C05484=1146.169,25.527,-49.640,179.957,6.278,149.150
C05485=1146.174,25.277,-49.625,179.955,6.277,149.150
C05486=1146.179,25.027,-49.611,179.952,6.277,149.151
C05487=1146.184,24.778,-49.597,179.949,6.275,149.151
C05488=1146.190,24.528,-49.582,179.947,6.275,149.152
C05489=1146.195,24.278,-49.568,179.945,6.274,149.152
C05490=1146.200,24.029,-49.554,179.941,6.272,149.153
C05491=1146.205,23.780,-49.539,179.939,6.272,149.154
C05492=1146.210,23.530,-49.525,179.937,6.271,149.154
C05493=1146.215,23.280,-49.510,179.934,6.270,149.155
C05494=1146.220,23.031,-49.496,179.932,6.269,149.155
C05495=1146.225,22.782,-49.482,179.929,6.268,149.156
C05496=1146.230,22.532,-49.468,179.927,6.267,149.156
C05497=1146.235,22.282,-49.454,179.924,6.266,149.157
C05498=1146.240,22.033,-49.439,179.921,6.265,149.157
C05499=1146.245,21.783,-49.425,179.919,6.265,149.158
C05500=1146.251,21.534,-49.411,179.916,6.263,149.159
C05501=1146.256,21.284,-49.397,179.914,6.262,149.159
C05502=1146.261,21.034,-49.382,179.911,6.262,149.160
C05503=1146.266,20.785,-49.368,179.908,6.260,149.160
C05504=1146.271,20.536,-49.354,179.906,6.260,149.161
C05505=1146.276,20.286,-49.340,179.904,6.259,149.161
C05506=1146.281,20.036,-49.326,179.901,6.257,149.162
C05507=1146.286,19.787,-49.311,179.898,6.257,149.162
C05508=1146.291,19.538,-49.298,179.896,6.256,149.163
C05509=1146.296,19.288,-49.283,179.893,6.256,149.164
C05510=1146.301,19.038,-49.269,179.891,6.254,149.164
C05511=1146.306,18.789,-49.255,179.888,6.253,149.164
C05512=1146.312,18.539,-49.241,179.886,6.253,149.165
C05513=1146.316,18.290,-49.227,179.883,6.251,149.166
C05514=1146.321,18.040,-49.214,179.880,6.251,149.166
C05515=1146.326,17.790,-49.199,179.878,6.250,149.167
C05516=1146.332,17.541,-49.185,179.876,6.250,149.167
C05517=1146.337,17.291,-49.171,179.873,6.248,149.168
C05518=1146.342,17.042,-49.157,179.871,6.247,149.168
C05519=1146.347,16.793,-49.143,179.868,6.247,149.169
C05520=1146.352,16.543,-49.129,179.865,6.245,149.169
C05521=1146.358,16.293,-49.115,179.863,6.245,149.170
C05522=1146.362,16.044,-49.102,179.860,6.244,149.171
C05523=1146.367,15.794,-49.087,179.858,6.243,149.171
C05524=1146.372,15.544,-49.073,179.855,6.242,149.172
C05525=1146.377,15.295,-49.059,179.853,6.241,149.172
C05526=1146.383,15.046,-49.045,179.850,6.240,149.173
C05527=1146.388,14.795,-49.031,179.848,6.240,149.173
C05528=1146.393,14.546,-49.017,179.845,6.238,149.174
C05529=1146.398,14.297,-49.004,179.843,6.238,149.174
C05530=1146.403,14.047,-48.990,179.840,6.237,149.175
C05531=1146.409,13.798,-48.976,179.838,6.236,149.176
C05532=1146.414,13.548,-48.962,179.835,6.235,149.176
C05533=1146.419,13.298,-48.948,179.832,6.234,149.177
C05534=1146.423,13.050,-48.935,179.830,6.233,149.177
C05535=1146.429,12.799,-48.921,179.827,6.233,149.178
C05536=1146.434,12.549,-48.907,179.825,6.231,149.178
C05537=1146.439,12.300,-48.893,179.822,6.231,149.179
C05538=1146.444,12.050,-48.879,179.820,6.230,149.180
C05539=1146.449,11.801,-48.866,179.818,6.229,149.180
C05540=1146.454,11.552,-48.852,179.814,6.228,149.181
C05541=1146.459,11.301,-48.838,179.812,6.227,149.181
C05542=1146.465,11.052,-48.824,179.810,6.227,149.182
C05543=1146.469,10.803,-48.810,179.807,6.226,149.182
C05544=1146.474,10.553,-48.797,179.804,6.225,149.183
C05545=1146.480,10.304,-48.783,179.802,6.224,149.183
C05546=1146.485,10.054,-48.770,179.799,6.223,149.184
C05547=1146.490,9.805,-48.756,179.797,6.223,149.185
C05548=1146.495,9.555,-48.742,179.794,6.221,149.185
C05549=1146.501,9.305,-48.729,179.792,6.221,149.186
C05550=1146.505,9.056,-48.715,179.790,6.220,149.186
C05551=1146.510,8.806,-48.701,179.787,6.219,149.187
C05552=1146.516,8.557,-48.687,179.785,6.218,149.187
C05553=1146.520,8.307,-48.675,179.782,6.217,149.188
C05554=1146.526,8.058,-48.661,179.779,6.216,149.188
C05555=1146.531,7.808,-48.646,179.777,6.216,149.189
C05556=1146.536,7.559,-48.634,179.775,6.215,149.190
C05557=1146.541,7.309,-48.619,179.772,6.214,149.190
C05558=1146.547,7.059,-48.606,179.769,6.213,149.191
C05559=1146.551,6.810,-48.593,179.767,6.212,149.191
C05560=1146.557,6.560,-48.579,179.764,6.212,149.192
C05561=1146.561,6.311,-48.566,179.762,6.211,149.192
C05562=1146.567,6.060,-48.552,179.759,6.209,149.193
C05563=1146.572,5.811,-48.538,179.757,6.209,149.194
C05564=1146.577,5.561,-48.525,179.754,6.208,149.194
C05565=1146.582,5.312,-48.512,179.752,6.208,149.195
C05566=1146.587,5.062,-48.498,179.750,6.207,149.195
C05567=1146.593,4.813,-48.485,179.746,6.206,149.196
C05568=1146.597,4.563,-48.471,179.744,6.205,149.196
C05569=1146.603,4.314,-48.458,179.742,6.204,149.197
C05570=1146.608,4.064,-48.444,179.739,6.204,149.197
C05571=1146.613,3.815,-48.431,179.737,6.203,149.198
C05572=1146.618,3.564,-48.418,179.734,6.202,149.199
C05573=1146.623,3.316,-48.405,179.732,6.201,149.199
C05574=1146.629,3.066,-48.391,179.729,6.200,149.200
C05575=1146.634,2.816,-48.378,179.727,6.199,149.200
C05576=1146.639,2.567,-48.364,179.724,6.199,149.201
C05577=1146.644,2.317,-48.351,179.722,6.198,149.201
C05578=1146.649,2.067,-48.338,179.719,6.197,149.202
C05579=1146.655,1.798,-48.323,179.717,6.196,149.202
C05580=1146.660,1.528,-48.309,179.714,6.196,149.203
C05581=1146.666,1.259,-48.295,179.711,6.194,149.204
C05582=1146.671,0.989,-48.281,179.709,6.194,149.204
C05583=1146.676,0.740,-48.267,179.706,6.193,149.205
C05584=1146.681,0.490,-48.254,179.704,6.192,149.205
C05585=1146.686,0.241,-48.241,179.701,6.191,149.206
C05586=1146.691,-0.009,-48.227,179.698,6.190,149.207
C05587=1146.697,-0.258,-48.214,179.696,6.190,149.207
C05588=1146.702,-0.508,-48.201,179.694,6.189,149.208
C05589=1146.707,-0.758,-48.188,179.691,6.188,149.208
C05590=1146.712,-1.007,-48.174,179.689,6.188,149.209
C05591=1146.717,-1.257,-48.161,179.686,6.186,149.209
C05592=1146.723,-1.506,-48.148,179.684,6.186,149.210
C05593=1146.727,-1.756,-48.135,179.681,6.185,149.211
C05594=1146.733,-2.006,-48.123,179.679,6.184,149.211
C05595=1146.738,-2.255,-48.109,179.676,6.184,149.212
C05596=1146.743,-2.505,-48.096,179.674,6.183,149.212
C05597=1146.748,-2.754,-48.082,179.671,6.183,149.213
C05598=1146.753,-3.004,-48.070,179.669,6.181,149.213
C05599=1146.758,-3.254,-48.057,179.666,6.180,149.214
C05600=1146.764,-3.503,-48.044,179.664,6.180,149.214
C05601=1146.769,-3.753,-48.031,179.662,6.179,149.215
C05602=1146.774,-4.002,-48.017,179.659,6.179,149.216
C05603=1146.779,-4.252,-48.004,179.657,6.178,149.216
C05604=1146.784,-4.502,-47.991,179.654,6.177,149.217
C05605=1146.790,-4.751,-47.978,179.651,6.176,149.217
C05606=1146.795,-5.000,-47.965,179.649,6.175,149.218
C05607=1146.799,-5.251,-47.953,179.647,6.174,149.218
C05608=1146.805,-5.500,-47.939,179.644,6.174,149.219
C05609=1146.810,-5.749,-47.927,179.642,6.173,149.220
C05610=1146.815,-5.999,-47.914,179.640,6.172,149.220
C05611=1146.821,-6.249,-47.901,179.637,6.172,149.221
C05612=1146.826,-6.498,-47.888,179.635,6.171,149.221
C05613=1146.830,-6.748,-47.875,179.631,6.170,149.222
C05614=1146.836,-6.998,-47.862,179.629,6.169,149.222
C05615=1146.841,-7.247,-47.849,179.627,6.168,149.223
C05616=1146.846,-7.497,-47.836,179.624,6.168,149.224
C05617=1146.852,-7.747,-47.823,179.622,6.167,149.224
C05618=1146.857,-7.996,-47.810,179.620,6.167,149.225
C05619=1146.861,-8.246,-47.797,179.617,6.166,149.225
C05620=1146.866,-8.496,-47.785,179.615,6.165,149.226
C05621=1146.872,-8.745,-47.772,179.612,6.164,149.226
C05622=1146.877,-8.995,-47.759,179.609,6.163,149.227
C05623=1146.882,-9.245,-47.746,179.607,6.163,149.227
C05624=1146.887,-9.494,-47.734,179.605,6.162,149.228
C05625=1146.893,-9.744,-47.720,179.602,6.161,149.229
C05626=1146.898,-9.993,-47.708,179.600,6.161,149.229
C05627=1146.903,-10.243,-47.695,179.597,6.160,149.230
C05628=1146.908,-10.492,-47.682,179.595,6.159,149.230
C05629=1146.913,-10.742,-47.670,179.593,6.159,149.231
C05630=1146.918,-10.992,-47.656,179.590,6.157,149.231
C05631=1146.923,-11.241,-47.643,179.587,6.157,149.232
C05632=1146.928,-11.491,-47.631,179.585,6.156,149.233
C05633=1146.934,-11.740,-47.619,179.583,6.155,149.233
C05634=1146.939,-11.990,-47.606,179.580,6.155,149.234
C05635=1146.944,-12.240,-47.593,179.578,6.154,149.234
C05636=1146.949,-12.489,-47.580,179.575,6.154,149.235
C05637=1146.954,-12.739,-47.568,179.573,6.153,149.235
C05638=1146.959,-12.988,-47.555,179.571,6.152,149.236
C05639=1146.964,-13.239,-47.543,179.568,6.152,149.237
C05640=1146.969,-13.488,-47.530,179.566,6.151,149.237
C05641=1146.975,-13.737,-47.517,179.564,6.150,149.238
C05642=1146.980,-13.987,-47.504,179.561,6.149,149.238
C05643=1146.986,-14.236,-47.492,179.558,6.148,149.239
C05644=1146.990,-14.487,-47.479,179.556,6.148,149.239
C05645=1146.995,-14.736,-47.467,179.553,6.147,149.240
C05646=1147.001,-14.986,-47.454,179.551,6.146,149.240
C05647=1147.006,-15.235,-47.442,179.549,6.145,149.241
C05648=1147.011,-15.485,-47.430,179.546,6.145,149.242
C05649=1147.016,-15.734,-47.417,179.544,6.144,149.242
C05650=1147.021,-15.984,-47.404,179.541,6.144,149.243
C05651=1147.027,-16.234,-47.391,179.539,6.143,149.243
C05652=1147.032,-16.484,-47.379,179.537,6.143,149.244
C05653=1147.037,-16.733,-47.366,179.534,6.142,149.244
C05654=1147.042,-16.982,-47.354,179.532,6.141,149.245
C05655=1147.048,-17.232,-47.342,179.530,6.141,149.246
C05656=1147.052,-17.482,-47.329,179.527,6.139,149.246
C05657=1147.057,-17.732,-47.316,179.524,6.139,149.247
C05658=1147.063,-17.982,-47.305,179.522,6.138,149.247
C05659=1147.068,-18.231,-47.292,179.519,6.137,149.248
C05660=1147.073,-18.480,-47.279,179.517,6.137,149.248
C05661=1147.079,-18.730,-47.267,179.514,6.136,149.249
C05662=1147.084,-18.979,-47.255,179.512,6.135,149.250
C05663=1147.089,-19.229,-47.242,179.510,6.135,149.250
C05664=1147.094,-19.479,-47.230,179.507,6.134,149.251
C05665=1147.099,-19.729,-47.217,179.505,6.133,149.251
C05666=1147.104,-19.979,-47.206,179.503,6.133,149.252
C05667=1147.109,-20.228,-47.193,179.500,6.132,149.252
C05668=1147.114,-20.477,-47.180,179.498,6.132,149.253
C05669=1147.120,-20.727,-47.168,179.496,6.131,149.254
C05670=1147.125,-20.977,-47.156,179.493,6.130,149.254
C05671=1147.130,-21.226,-47.144,179.491,6.130,149.255
C05672=1147.136,-21.476,-47.131,179.488,6.129,149.255
C05673=1147.141,-21.726,-47.119,179.486,6.128,149.256
C05674=1147.146,-21.975,-47.107,179.484,6.128,149.256
C05675=1147.151,-22.225,-47.095,179.481,6.127,149.257
C05676=1147.156,-22.475,-47.082,179.479,6.126,149.258
C05677=1147.161,-22.725,-47.070,179.477,6.126,149.258
C05678=1147.167,-22.974,-47.058,179.474,6.125,149.259
C05679=1147.172,-23.224,-47.046,179.472,6.124,149.259
C05680=1147.177,-23.474,-47.033,179.469,6.123,149.260
C05681=1147.183,-23.723,-47.021,179.466,6.122,149.260
C05682=1147.187,-23.972,-47.009,179.464,6.122,149.261
C05683=1147.194,-24.242,-46.996,179.461,6.121,149.261
C05684=1147.199,-24.513,-46.983,179.459,6.121,149.262
C05685=1147.204,-24.783,-46.970,179.456,6.120,149.263
C05686=1147.210,-25.052,-46.957,179.454,6.120,149.263
C05687=1147.215,-25.302,-46.945,179.451,6.119,149.264
C05688=1147.220,-25.551,-46.932,179.449,6.118,149.265
C05689=1147.226,-25.801,-46.920,179.447,6.118,149.265
C05690=1147.231,-26.051,-46.908,179.444,6.117,149.266
C05691=1147.236,-26.301,-46.896,179.442,6.116,149.266
C05692=1147.241,-26.550,-46.885,179.439,6.116,149.267
C05693=1147.246,-26.800,-46.872,179.437,6.115,149.267
C05694=1147.252,-27.049,-46.860,179.435,6.115,149.268
C05695=1147.257,-27.299,-46.848,179.432,6.114,149.268
C05696=1147.262,-27.549,-46.836,179.430,6.113,149.269
C05697=1147.268,-27.799,-46.824,179.428,6.113,149.270
C05698=1147.272,-28.048,-46.812,179.425,6.112,149.270
C05699=1147.277,-28.298,-46.800,179.423,6.112,149.271
C05700=1147.283,-28.548,-46.788,179.421,6.111,149.271
C05701=1147.288,-28.797,-46.776,179.418,6.110,149.272
C05702=1147.293,-29.047,-46.763,179.416,6.110,149.272
C05703=1147.298,-29.296,-46.752,179.414,6.109,149.273
C05704=1147.303,-29.546,-46.740,179.411,6.108,149.274
C05705=1147.309,-29.796,-46.728,179.409,6.108,149.274
C05706=1147.314,-30.046,-46.716,179.406,6.107,149.275
C05707=1147.319,-30.295,-46.704,179.404,6.106,149.275
C05708=1147.324,-30.545,-46.693,179.401,6.106,149.276
C05709=1147.330,-30.795,-46.681,179.399,6.105,149.276
C05710=1147.335,-31.044,-46.668,179.397,6.104,149.277
C05711=1147.339,-31.294,-46.657,179.394,6.104,149.278
C05712=1147.345,-31.544,-46.645,179.392,6.103,149.278
C05713=1147.350,-31.794,-46.633,179.389,6.103,149.279
C05714=1147.355,-32.043,-46.620,179.387,6.102,149.279
C05715=1147.360,-32.293,-46.609,179.385,6.101,149.280
C05716=1147.366,-32.542,-46.598,179.382,6.101,149.280
C05717=1147.372,-32.792,-46.586,179.380,6.100,149.281
C05718=1147.376,-33.042,-46.574,179.377,6.100,149.282
C05719=1147.382,-33.292,-46.563,179.375,6.099,149.282
C05720=1147.387,-33.541,-46.550,179.373,6.098,149.283
C05721=1147.391,-33.791,-46.539,179.370,6.098,149.283
C05722=1147.397,-34.041,-46.527,179.368,6.097,149.284
C05723=1147.402,-34.290,-46.515,179.366,6.096,149.284
C05724=1147.407,-34.540,-46.504,179.363,6.096,149.285
C05725=1147.413,-34.789,-46.492,179.361,6.095,149.286
C05726=1147.418,-35.039,-46.480,179.358,6.094,149.286
C05727=1147.423,-35.288,-46.468,179.356,6.094,149.287
C05728=1147.428,-35.538,-46.456,179.354,6.093,149.287
C05729=1147.434,-35.788,-46.444,179.352,6.093,149.288
C05730=1147.438,-36.038,-46.433,179.349,6.093,149.288
C05731=1147.444,-36.288,-46.421,179.347,6.092,149.289
C05732=1147.450,-36.537,-46.410,179.345,6.092,149.290
C05733=1147.455,-36.787,-46.398,179.342,6.091,149.290
C05734=1147.460,-37.036,-46.387,179.340,6.090,149.291
C05735=1147.465,-37.286,-46.375,179.337,6.090,149.291
C05736=1147.470,-37.536,-46.363,179.335,6.089,149.292
C05737=1147.476,-37.786,-46.352,179.333,6.088,149.292
C05738=1147.481,-38.035,-46.341,179.330,6.088,149.293
C05739=1147.486,-38.285,-46.329,179.328,6.087,149.293
C05740=1147.491,-38.534,-46.317,179.326,6.086,149.294
C05741=1147.496,-38.784,-46.306,179.323,6.086,149.295
C05742=1147.502,-39.034,-46.294,179.321,6.085,149.295
C05743=1147.507,-39.283,-46.283,179.319,6.084,149.296
C05744=1147.513,-39.533,-46.271,179.316,6.084,149.296
C05745=1147.517,-39.783,-46.260,179.314,6.083,149.297
C05746=1147.523,-40.033,-46.248,179.312,6.083,149.297
C05747=1147.527,-40.282,-46.236,179.309,6.083,149.298
C05748=1147.533,-40.532,-46.225,179.307,6.082,149.299
C05749=1147.538,-40.781,-46.214,179.305,6.082,149.299
C05750=1147.544,-41.031,-46.202,179.302,6.081,149.300
C05751=1147.549,-41.281,-46.190,179.300,6.080,149.300
C05752=1147.554,-41.531,-46.179,179.298,6.080,149.301
C05753=1147.560,-41.781,-46.168,179.295,6.079,149.301
C05754=1147.565,-42.030,-46.156,179.293,6.078,149.302
C05755=1147.570,-42.280,-46.145,179.291,6.078,149.303
C05756=1147.575,-42.530,-46.133,179.288,6.077,149.303
C05757=1147.580,-42.779,-46.122,179.286,6.076,149.304
C05758=1147.586,-43.029,-46.110,179.284,6.076,149.304
C05759=1147.590,-43.278,-46.099,179.281,6.076,149.305
C05760=1147.596,-43.528,-46.087,179.279,6.075,149.305
C05761=1147.601,-43.778,-46.077,179.277,6.074,149.306
C05762=1147.607,-44.028,-46.065,179.274,6.074,149.307
C05763=1147.611,-44.277,-46.054,179.272,6.073,149.307
C05764=1147.617,-44.527,-46.042,179.270,6.073,149.308
C05765=1147.622,-44.776,-46.031,179.267,6.072,149.308
C05766=1147.628,-45.027,-46.020,179.265,6.071,149.309
C05767=1147.633,-45.276,-46.009,179.262,6.071,149.309
C05768=1147.638,-45.525,-45.998,179.261,6.071,149.310
C05769=1147.643,-45.775,-45.986,179.258,6.071,149.311
C05770=1147.648,-46.025,-45.975,179.256,6.070,149.311
C05771=1147.654,-46.275,-45.963,179.254,6.069,149.312
C05772=1147.659,-46.524,-45.952,179.251,6.069,149.312
C05773=1147.664,-46.774,-45.941,179.249,6.068,149.313
C05774=1147.669,-47.024,-45.929,179.246,6.067,149.313
C05775=1147.675,-47.273,-45.919,179.244,6.067,149.314
C05776=1147.680,-47.523,-45.907,179.242,6.066,149.314
C05777=1147.685,-47.773,-45.896,179.240,6.066,149.315
C05778=1147.690,-48.022,-45.885,179.238,6.065,149.316
C05779=1147.696,-48.272,-45.874,179.236,6.065,149.316
C05780=1147.701,-48.522,-45.862,179.233,6.064,149.317
C05781=1147.706,-48.771,-45.852,179.231,6.063,149.317
C05782=1147.712,-49.022,-45.840,179.228,6.063,149.318
C05783=1147.716,-49.271,-45.829,179.226,6.062,149.318
C05784=1147.722,-49.520,-45.818,179.224,6.061,149.319
C05785=1147.727,-49.771,-45.807,179.221,6.061,149.320
C05786=1147.732,-50.020,-45.796,179.219,6.061,149.320
C05787=1147.738,-50.291,-45.784,179.217,6.061,149.321
C05788=1147.744,-50.562,-45.772,179.215,6.060,149.321
C05789=1147.749,-50.833,-45.759,179.212,6.060,149.322
C05790=1147.755,-51.103,-45.748,179.209,6.059,149.323
C05791=1147.760,-51.352,-45.736,179.207,6.058,149.323
C05792=1147.765,-51.603,-45.726,179.205,6.058,149.324
C05793=1147.771,-51.852,-45.715,179.202,6.057,149.324
C05794=1147.776,-52.102,-45.703,179.200,6.056,149.325
C05795=1147.782,-52.351,-45.693,179.198,6.056,149.325
C05796=1147.786,-52.601,-45.681,179.195,6.055,149.326
C05797=1147.791,-52.851,-45.671,179.194,6.055,149.326
C05798=1147.797,-53.100,-45.659,179.191,6.055,149.327
C05799=1147.802,-53.350,-45.649,179.189,6.054,149.328
C05800=1147.808,-53.599,-45.638,179.186,6.053,149.328
C05801=1147.813,-53.850,-45.627,179.184,6.053,149.329
C05802=1147.818,-54.100,-45.615,179.182,6.052,149.329
C05803=1147.824,-54.349,-45.605,179.179,6.052,149.330
C05804=1147.828,-54.599,-45.594,179.177,6.052,149.330
C05805=1147.834,-54.848,-45.584,179.175,6.051,149.331
C05806=1147.839,-55.098,-45.572,179.172,6.051,149.332
C05807=1147.844,-55.348,-45.561,179.170,6.050,149.332
C05808=1147.850,-55.597,-45.550,179.168,6.049,149.333
C05809=1147.855,-55.848,-45.540,179.165,6.049,149.333
C05810=1147.860,-56.097,-45.529,179.163,6.048,149.334
C05811=1147.865,-56.347,-45.518,179.161,6.048,149.335
C05812=1147.870,-56.596,-45.507,179.159,6.047,149.335
C05813=1147.876,-56.846,-45.496,179.157,6.047,149.335
C05814=1147.881,-57.096,-45.485,179.154,6.046,149.336
C05815=1147.886,-57.345,-45.474,179.152,6.045,149.337
C05816=1147.891,-57.596,-45.464,179.150,6.045,149.337
C05817=1147.897,-57.845,-45.453,179.148,6.045,149.338
C05818=1147.902,-58.095,-45.442,179.146,6.044,149.338
C05819=1147.908,-58.344,-45.431,179.143,6.044,149.339
C05820=1147.913,-58.594,-45.420,179.141,6.043,149.340
C05821=1147.918,-58.844,-45.410,179.138,6.042,149.340
C05822=1147.923,-59.093,-45.399,179.136,6.043,149.341
C05823=1147.928,-59.343,-45.389,179.134,6.042,149.341
C05824=1147.933,-59.593,-45.377,179.132,6.041,149.342
C05825=1147.939,-59.842,-45.367,179.129,6.041,149.342
C05826=1147.944,-60.092,-45.357,179.127,6.040,149.343
C05827=1147.949,-60.341,-45.346,179.125,6.039,149.343
C05828=1147.955,-60.592,-45.334,179.123,6.040,149.344
C05829=1147.960,-60.841,-45.324,179.121,6.039,149.344
C05830=1147.965,-61.091,-45.313,179.118,6.039,149.345
C05831=1147.971,-61.341,-45.303,179.116,6.038,149.346
C05832=1147.976,-61.591,-45.292,179.114,6.037,149.346
C05833=1147.981,-61.840,-45.281,179.112,6.037,149.347
C05834=1147.986,-62.090,-45.271,179.109,6.037,149.347
C05835=1147.992,-62.340,-45.260,179.107,6.036,149.348
C05836=1147.997,-62.590,-45.250,179.105,6.035,149.349
C05837=1148.002,-62.839,-45.239,179.102,6.035,149.349
C05838=1148.007,-63.089,-45.228,179.101,6.035,149.349
C05839=1148.012,-63.339,-45.218,179.098,6.034,149.350
C05840=1148.017,-63.589,-45.208,179.096,6.033,149.351
C05841=1148.023,-63.838,-45.197,179.094,6.033,149.351
C05842=1148.028,-64.088,-45.186,179.091,6.032,149.352
C05843=1148.033,-64.338,-45.176,179.089,6.032,149.352
C05844=1148.039,-64.587,-45.166,179.087,6.032,149.353
C05845=1148.044,-64.837,-45.154,179.085,6.031,149.354
C05846=1148.049,-65.086,-45.144,179.082,6.030,149.354
C05847=1148.054,-65.336,-45.134,179.080,6.030,149.355
C05848=1148.060,-65.586,-45.123,179.078,6.030,149.355
C05849=1148.065,-65.836,-45.113,179.076,6.029,149.356
C05850=1148.070,-66.085,-45.102,179.073,6.029,149.356
C05851=1148.076,-66.335,-45.092,179.071,6.028,149.357
C05852=1148.081,-66.585,-45.081,179.069,6.028,149.357
C05853=1148.086,-66.835,-45.071,179.067,6.028,149.358
C05854=1148.091,-67.085,-45.060,179.065,6.027,149.359
C05855=1148.097,-67.334,-45.050,179.062,6.026,149.359
C05856=1148.103,-67.584,-45.040,179.060,6.026,149.360
C05857=1148.107,-67.833,-45.029,179.058,6.026,149.360
C05858=1148.113,-68.083,-45.018,179.056,6.025,149.361
C05859=1148.118,-68.333,-45.008,179.053,6.025,149.361
C05860=1148.123,-68.583,-44.998,179.051,6.024,149.362
C05861=1148.129,-68.832,-44.987,179.050,6.024,149.362
C05862=1148.134,-69.083,-44.977,179.047,6.024,149.363
C05863=1148.140,-69.332,-44.967,179.045,6.023,149.364
C05864=1148.145,-69.582,-44.956,179.042,6.022,149.364
C05865=1148.149,-69.832,-44.946,179.040,6.022,149.365
C05866=1148.155,-70.081,-44.936,179.038,6.022,149.365
C05867=1148.160,-70.331,-44.926,179.036,6.021,149.366
C05868=1148.166,-70.581,-44.915,179.033,6.020,149.366
C05869=1148.171,-70.830,-44.905,179.031,6.020,149.367
C05870=1148.176,-71.080,-44.894,179.030,6.020,149.367
C05871=1148.182,-71.330,-44.884,179.027,6.019,149.368
C05872=1148.187,-71.579,-44.874,179.025,6.019,149.369
C05873=1148.192,-71.829,-44.863,179.023,6.018,149.369
C05874=1148.197,-72.079,-44.853,179.020,6.018,149.370
C05875=1148.203,-72.328,-44.843,179.018,6.017,149.370
C05876=1148.208,-72.578,-44.833,179.016,6.017,149.371
C05877=1148.213,-72.828,-44.822,179.013,6.016,149.371
C05878=1148.219,-73.078,-44.813,179.012,6.016,149.372
C05879=1148.224,-73.328,-44.802,179.010,6.016,149.372
C05880=1148.230,-73.578,-44.792,179.007,6.015,149.373
C05881=1148.235,-73.827,-44.782,179.005,6.014,149.374
C05882=1148.240,-74.077,-44.772,179.003,6.014,149.374
C05883=1148.245,-74.327,-44.762,179.000,6.014,149.375
C05884=1148.251,-74.577,-44.751,178.998,6.013,149.375
C05885=1148.256,-74.826,-44.741,178.996,6.012,149.376
C05886=1148.261,-75.076,-44.731,178.994,6.013,149.376
C05887=1148.266,-75.326,-44.721,178.992,6.012,149.377
C05888=1148.272,-75.575,-44.711,178.990,6.011,149.377
C05889=1148.277,-75.825,-44.701,178.987,6.011,149.378
C05890=1148.282,-76.075,-44.690,178.985,6.011,149.379
C05891=1148.288,-76.346,-44.680,178.983,6.010,149.379
C05892=1148.294,-76.618,-44.669,178.980,6.010,149.380
C05893=1148.300,-76.889,-44.658,178.978,6.009,149.380
C05894=1148.305,-77.160,-44.647,178.976,6.009,149.381
C05895=1148.310,-77.410,-44.637,178.973,6.008,149.381
C05896=1148.316,-77.660,-44.627,178.972,6.008,149.382
C05897=1148.322,-77.910,-44.617,178.969,6.008,149.383
C05898=1148.327,-78.159,-44.607,178.967,6.007,149.383
C05899=1148.332,-78.409,-44.597,178.965,6.007,149.384
C05900=1148.337,-78.659,-44.586,178.963,6.006,149.384
C05901=1148.343,-78.909,-44.577,178.961,6.006,149.385
C05902=1148.348,-79.158,-44.567,178.958,6.005,149.385
C05903=1148.353,-79.408,-44.557,178.956,6.005,149.386
C05904=1148.359,-79.658,-44.547,178.954,6.005,149.386
C05905=1148.364,-79.907,-44.536,178.952,6.004,149.387
C05906=1148.369,-80.157,-44.527,178.950,6.004,149.388
C05907=1148.374,-80.407,-44.517,178.948,6.003,149.388
C05908=1148.380,-80.657,-44.507,178.945,6.003,149.389
C05909=1148.385,-80.906,-44.497,178.943,6.002,149.389
C05910=1148.391,-81.156,-44.488,178.941,6.002,149.390
C05911=1148.396,-81.406,-44.477,178.939,6.002,149.390
C05912=1148.401,-81.656,-44.467,178.937,6.001,149.391
C05913=1148.406,-81.905,-44.457,178.935,6.001,149.391
C05914=1148.412,-82.156,-44.448,178.932,6.000,149.392
C05915=1148.417,-82.405,-44.438,178.930,6.000,149.392
C05916=1148.423,-82.654,-44.428,178.928,5.999,149.393
C05917=1148.428,-82.905,-44.418,178.926,5.999,149.394
C05918=1148.433,-83.154,-44.408,178.924,5.999,149.394
C05919=1148.438,-83.404,-44.398,178.922,5.998,149.395
C05920=1148.443,-83.653,-44.389,178.920,5.998,149.395
C05921=1148.449,-83.903,-44.379,178.917,5.997,149.396
C05922=1148.455,-84.153,-44.369,178.915,5.997,149.396
C05923=1148.459,-84.403,-44.359,178.914,5.997,149.397
C05924=1148.465,-84.653,-44.349,178.911,5.996,149.397
C05925=1148.471,-84.902,-44.339,178.909,5.996,149.398
C05926=1148.476,-85.152,-44.330,178.907,5.996,149.398
C05927=1148.481,-85.402,-44.320,178.904,5.995,149.399
C05928=1148.486,-85.651,-44.310,178.902,5.994,149.400
C05929=1148.491,-85.902,-44.301,178.900,5.994,149.400
C05930=1148.496,-86.151,-44.291,178.898,5.994,149.401
C05931=1148.502,-86.401,-44.281,178.896,5.993,149.401
C05932=1148.508,-86.651,-44.271,178.894,5.993,149.402
C05933=1148.513,-86.900,-44.262,178.892,5.993,149.402
C05934=1148.519,-87.150,-44.252,178.889,5.992,149.403
C05935=1148.523,-87.400,-44.243,178.887,5.991,149.403
C05936=1148.529,-87.650,-44.233,178.886,5.991,149.404
C05937=1148.534,-87.900,-44.223,178.883,5.991,149.404
C05938=1148.539,-88.149,-44.213,178.881,5.990,149.405
C05939=1148.544,-88.399,-44.204,178.879,5.990,149.406
C05940=1148.550,-88.649,-44.194,178.877,5.990,149.406
C05941=1148.555,-88.898,-44.185,178.875,5.989,149.407
C05942=1148.561,-89.148,-44.175,178.873,5.989,149.407
C05943=1148.566,-89.398,-44.166,178.870,5.988,149.408
C05944=1148.571,-89.647,-44.156,178.868,5.988,149.408
C05945=1148.576,-89.898,-44.146,178.867,5.988,149.409
C05946=1148.582,-90.147,-44.136,178.864,5.987,149.409
C05947=1148.587,-90.397,-44.127,178.862,5.987,149.410
C05948=1148.592,-90.647,-44.117,178.860,5.987,149.410
C05949=1148.598,-90.897,-44.108,178.858,5.986,149.411
C05950=1148.603,-91.146,-44.098,178.855,5.986,149.412
C05951=1148.608,-91.396,-44.089,178.854,5.986,149.412
C05952=1148.614,-91.646,-44.079,178.852,5.985,149.413
C05953=1148.619,-91.895,-44.070,178.849,5.984,149.413
C05954=1148.625,-92.145,-44.060,178.847,5.984,149.414
C05955=1148.630,-92.395,-44.051,178.845,5.984,149.414
C05956=1148.636,-92.645,-44.041,178.843,5.983,149.415
C05957=1148.641,-92.894,-44.032,178.841,5.983,149.415
C05958=1148.646,-93.144,-44.023,178.839,5.983,149.416
C05959=1148.651,-93.394,-44.012,178.836,5.982,149.416
C05960=1148.656,-93.644,-44.003,178.835,5.982,149.417
C05961=1148.662,-93.894,-43.994,178.832,5.981,149.418
C05962=1148.667,-94.144,-43.984,178.831,5.982,149.418
C05963=1148.673,-94.394,-43.975,178.828,5.981,149.419
C05964=1148.678,-94.643,-43.965,178.826,5.980,149.419
C05965=1148.683,-94.893,-43.956,178.824,5.980,149.420
C05966=1148.689,-95.143,-43.947,178.822,5.980,149.420
C05967=1148.693,-95.392,-43.937,178.820,5.979,149.421
C05968=1148.699,-95.642,-43.928,178.818,5.979,149.421
C05969=1148.705,-95.892,-43.919,178.816,5.978,149.422
C05970=1148.709,-96.142,-43.909,178.813,5.978,149.422
C05971=1148.715,-96.392,-43.900,178.812,5.978,149.423
C05972=1148.720,-96.642,-43.891,178.809,5.977,149.423
C05973=1148.725,-96.891,-43.881,178.808,5.977,149.424
C05974=1148.731,-97.141,-43.872,178.805,5.977,149.425
C05975=1148.736,-97.391,-43.863,178.803,5.976,149.425
C05976=1148.742,-97.640,-43.852,178.801,5.976,149.426
C05977=1148.747,-97.890,-43.844,178.799,5.975,149.426
C05978=1148.752,-98.140,-43.835,178.796,5.975,149.427
C05979=1148.758,-98.390,-43.825,178.795,5.975,149.427
C05980=1148.763,-98.639,-43.816,178.793,5.974,149.428
C05981=1148.768,-98.889,-43.807,178.791,5.973,149.428
C05982=1148.774,-99.139,-43.797,178.789,5.973,149.429
C05983=1148.779,-99.389,-43.788,178.786,5.973,149.429
C05984=1148.784,-99.639,-43.779,178.785,5.973,149.430
C05985=1148.791,-99.888,-43.770,178.782,5.972,149.430
C05986=1148.796,-100.138,-43.761,178.780,5.972,149.431
C05987=1148.801,-100.388,-43.752,178.778,5.972,149.432
C05988=1148.806,-100.637,-43.742,178.776,5.971,149.432
C05989=1148.812,-100.887,-43.733,178.774,5.971,149.433
C05990=1148.817,-101.137,-43.724,178.772,5.971,149.433
C05991=1148.822,-101.387,-43.715,178.770,5.970,149.434
C05992=1148.828,-101.636,-43.705,178.768,5.970,149.434
C05993=1148.833,-101.886,-43.696,178.766,5.969,149.435
C05994=1148.838,-102.136,-43.687,178.764,5.969,149.435
C05995=1148.844,-102.409,-43.677,178.762,5.969,149.436
C05996=1148.849,-102.680,-43.667,178.759,5.968,149.436
C05997=1148.855,-102.952,-43.657,178.757,5.968,149.437
C05998=1148.862,-103.225,-43.647,178.754,5.967,149.438
C05999=1148.867,-103.474,-43.638,178.753,5.967,149.438
C06000=1148.872,-103.724,-43.629,178.751,5.966,149.439
C06001=1148.877,-103.973,-43.620,178.749,5.967,149.439
C06002=1148.882,-104.223,-43.611,178.747,5.966,149.440
C06003=1148.888,-104.474,-43.601,178.744,5.965,149.440
C06004=1148.893,-104.723,-43.592,178.743,5.965,149.441
C06005=1148.899,-104.973,-43.584,178.740,5.965,149.441
C06006=1148.904,-105.223,-43.575,178.739,5.965,149.442
C06007=1148.909,-105.472,-43.566,178.737,5.964,149.442
C06008=1148.915,-105.722,-43.557,178.734,5.964,149.443
C06009=1148.920,-105.972,-43.547,178.732,5.964,149.443
C06010=1148.925,-106.221,-43.538,178.730,5.963,149.444
C06011=1148.931,-106.471,-43.529,178.728,5.963,149.444
C06012=1148.936,-106.721,-43.520,178.726,5.962,149.445
C06013=1148.942,-106.971,-43.511,178.724,5.963,149.446
C06014=1148.947,-107.221,-43.502,178.722,5.962,149.446
C06015=1148.953,-107.470,-43.493,178.720,5.961,149.447
C06016=1148.958,-107.720,-43.485,178.718,5.961,149.447
C06017=1148.963,-107.970,-43.476,178.716,5.960,149.448
C06018=1148.968,-108.220,-43.467,178.714,5.960,149.448
C06019=1148.973,-108.470,-43.458,178.712,5.960,149.449
C06020=1148.979,-108.720,-43.448,178.710,5.959,149.449
C06021=1148.984,-108.970,-43.439,178.708,5.959,149.450
C06022=1148.990,-109.219,-43.431,178.706,5.959,149.450
C06023=1148.995,-109.469,-43.422,178.704,5.959,149.451
C06024=1149.000,-109.719,-43.413,178.702,5.958,149.451
C06025=1149.006,-109.968,-43.404,178.700,5.958,149.452
C06026=1149.011,-110.218,-43.395,178.698,5.958,149.452
C06027=1149.016,-110.468,-43.386,178.695,5.957,149.453
C06028=1149.022,-110.718,-43.377,178.694,5.957,149.453
C06029=1149.028,-110.967,-43.368,178.692,5.956,149.454
C06030=1149.033,-111.217,-43.359,178.690,5.956,149.455
C06031=1149.038,-111.467,-43.351,178.687,5.956,149.455
C06032=1149.043,-111.717,-43.342,178.686,5.956,149.456
C06033=1149.049,-111.967,-43.334,178.684,5.955,149.456
C06034=1149.054,-112.217,-43.325,178.681,5.954,149.457
C06035=1149.060,-112.466,-43.316,178.680,5.954,149.457
C06036=1149.065,-112.716,-43.307,178.678,5.954,149.458
C06037=1149.070,-112.966,-43.298,178.676,5.954,149.458
C06038=1149.076,-113.215,-43.290,178.673,5.953,149.459
C06039=1149.081,-113.465,-43.281,178.672,5.953,149.459
C06040=1149.086,-113.715,-43.272,178.670,5.952,149.460
C06041=1149.092,-113.965,-43.262,178.668,5.953,149.460
C06042=1149.097,-114.215,-43.254,178.666,5.952,149.461
C06043=1149.103,-114.465,-43.246,178.663,5.951,149.461
C06044=1149.108,-114.715,-43.237,178.662,5.951,149.462
C06045=1149.113,-114.965,-43.228,178.659,5.951,149.462
C06046=1149.119,-115.214,-43.219,178.658,5.951,149.463
C06047=1149.124,-115.464,-43.211,178.656,5.950,149.463
C06048=1149.130,-115.713,-43.202,178.654,5.950,149.464
C06049=1149.135,-115.964,-43.193,178.652,5.949,149.464
C06050=1149.140,-116.214,-43.185,178.650,5.950,149.465
C06051=1149.146,-116.463,-43.176,178.647,5.949,149.465
C06052=1149.151,-116.713,-43.167,178.645,5.948,149.466
C06053=1149.156,-116.963,-43.158,178.644,5.948,149.466
C06054=1149.162,-117.213,-43.150,178.641,5.947,149.467
C06055=1149.167,-117.462,-43.141,178.640,5.948,149.467
C06056=1149.173,-117.712,-43.133,178.638,5.947,149.468
C06057=1149.178,-117.962,-43.124,178.636,5.947,149.468
C06058=1149.183,-118.212,-43.116,178.633,5.946,149.469
C06059=1149.189,-118.461,-43.107,178.632,5.947,149.470
C06060=1149.194,-118.711,-43.098,178.630,5.946,149.470
C06061=1149.199,-118.961,-43.089,178.628,5.946,149.471
C06062=1149.204,-119.210,-43.081,178.626,5.945,149.471
C06063=1149.210,-119.461,-43.073,178.624,5.945,149.472
C06064=1149.215,-119.710,-43.064,178.622,5.944,149.472
C06065=1149.220,-119.960,-43.055,178.620,5.944,149.473
C06066=1149.226,-120.210,-43.047,178.618,5.944,149.473
C06067=1149.231,-120.460,-43.039,178.616,5.943,149.474
C06068=1149.237,-120.710,-43.030,178.614,5.943,149.474
C06069=1149.242,-120.959,-43.021,178.612,5.943,149.475
C06070=1149.248,-121.209,-43.013,178.610,5.943,149.475
C06071=1149.253,-121.459,-43.004,178.608,5.942,149.476
C06072=1149.259,-121.708,-42.996,178.606,5.942,149.476
C06073=1149.264,-121.959,-42.987,178.604,5.941,149.477
C06074=1149.269,-122.208,-42.979,178.603,5.941,149.477
C06075=1149.274,-122.457,-42.971,178.600,5.941,149.478
C06076=1149.280,-122.708,-42.962,178.598,5.941,149.478
C06077=1149.285,-122.958,-42.953,178.596,5.940,149.479
C06078=1149.291,-123.207,-42.945,178.595,5.940,149.479
C06079=1149.296,-123.457,-42.937,178.592,5.939,149.480
C06080=1149.302,-123.707,-42.928,178.591,5.939,149.480
C06081=1149.308,-123.957,-42.920,178.589,5.939,149.481
C06082=1149.312,-124.207,-42.912,178.587,5.939,149.481
C06083=1149.317,-124.456,-42.903,178.585,5.938,149.482
C06084=1149.323,-124.706,-42.895,178.583,5.938,149.482
C06085=1149.328,-124.956,-42.886,178.581,5.937,149.483
C06086=1149.334,-125.207,-42.878,178.579,5.938,149.483
C06087=1149.340,-125.456,-42.869,178.577,5.937,149.484
C06088=1149.344,-125.705,-42.861,178.575,5.937,149.484
C06089=1149.350,-125.956,-42.853,178.573,5.936,149.485
C06090=1149.355,-126.205,-42.844,178.571,5.936,149.485
C06091=1149.361,-126.455,-42.836,178.569,5.936,149.486
C06092=1149.367,-126.704,-42.828,178.567,5.936,149.486
C06093=1149.371,-126.955,-42.820,178.565,5.935,149.487
C06094=1149.376,-127.204,-42.811,178.564,5.935,149.487
C06095=1149.382,-127.454,-42.803,178.561,5.934,149.488
C06096=1149.388,-127.704,-42.794,178.560,5.934,149.488
C06097=1149.393,-127.954,-42.786,178.558,5.933,149.489
C06098=1149.399,-128.204,-42.778,178.556,5.934,149.490
C06099=1148.977,-128.215,-42.821,178.552,5.937,149.491
C06100=1148.973,-127.965,-42.829,178.554,5.937,149.491
C06101=1148.967,-127.715,-42.837,178.556,5.937,149.490
C06102=1148.961,-127.466,-42.846,178.558,5.937,149.490
C06103=1148.956,-127.215,-42.854,178.560,5.938,149.489
C06104=1148.950,-126.966,-42.862,178.561,5.938,149.489
C06105=1148.945,-126.716,-42.870,178.564,5.939,149.488
C06106=1148.940,-126.466,-42.879,178.565,5.939,149.488
C06107=1148.934,-126.216,-42.887,178.567,5.940,149.487
C06108=1148.929,-125.966,-42.896,178.569,5.940,149.487
C06109=1148.923,-125.716,-42.904,178.571,5.940,149.486
C06110=1148.918,-125.467,-42.912,178.574,5.941,149.486
C06111=1148.913,-125.217,-42.921,178.575,5.941,149.485
C06112=1148.907,-124.968,-42.929,178.578,5.941,149.485
C06113=1148.902,-124.718,-42.937,178.579,5.941,149.484
C06114=1148.897,-124.467,-42.946,178.581,5.942,149.484
C06115=1148.891,-124.218,-42.954,178.583,5.942,149.483
C06116=1148.886,-123.968,-42.963,178.585,5.943,149.483
C06117=1148.881,-123.718,-42.971,178.587,5.943,149.482
C06118=1148.875,-123.469,-42.979,178.589,5.943,149.482
C06119=1148.870,-123.218,-42.987,178.591,5.943,149.481
C06120=1148.864,-122.969,-42.996,178.593,5.944,149.481
C06121=1148.859,-122.719,-43.005,178.595,5.944,149.480
C06122=1148.853,-122.469,-43.013,178.597,5.944,149.479
C06123=1148.848,-122.219,-43.022,178.599,5.944,149.479
C06124=1148.842,-121.970,-43.030,178.601,5.945,149.478
C06125=1148.838,-121.720,-43.038,178.603,5.945,149.478
C06126=1148.832,-121.470,-43.047,178.605,5.946,149.477
C06127=1148.827,-121.221,-43.055,178.606,5.946,149.477
C06128=1148.821,-120.970,-43.064,178.609,5.947,149.477
C06129=1148.816,-120.720,-43.072,178.610,5.947,149.476
C06130=1148.810,-120.471,-43.081,178.612,5.947,149.476
C06131=1148.805,-120.221,-43.090,178.614,5.947,149.475
C06132=1148.800,-119.971,-43.098,178.617,5.948,149.474
C06133=1148.794,-119.721,-43.107,178.618,5.948,149.474
C06134=1148.789,-119.472,-43.116,178.620,5.948,149.473
C06135=1148.783,-119.222,-43.124,178.623,5.949,149.473
C06136=1148.778,-118.972,-43.133,178.624,5.949,149.472
C06137=1148.773,-118.723,-43.141,178.626,5.950,149.472
C06138=1148.768,-118.473,-43.149,178.628,5.950,149.471
C06139=1148.762,-118.223,-43.158,178.631,5.950,149.471
C06140=1148.757,-117.973,-43.167,178.632,5.950,149.470
C06141=1148.751,-117.724,-43.175,178.634,5.951,149.470
C06142=1148.746,-117.474,-43.184,178.636,5.951,149.469
C06143=1148.741,-117.223,-43.192,178.638,5.952,149.469
C06144=1148.736,-116.973,-43.201,178.640,5.952,149.468
C06145=1148.730,-116.724,-43.210,178.642,5.952,149.468
C06146=1148.725,-116.474,-43.218,178.644,5.952,149.467
C06147=1148.720,-116.225,-43.227,178.646,5.953,149.467
C06148=1148.714,-115.974,-43.236,178.648,5.953,149.466
C06149=1148.708,-115.725,-43.244,178.650,5.953,149.466
C06150=1148.703,-115.475,-43.253,178.652,5.954,149.465
C06151=1148.698,-115.225,-43.262,178.654,5.954,149.465
C06152=1148.693,-114.975,-43.271,178.656,5.955,149.464
C06153=1148.687,-114.726,-43.279,178.658,5.955,149.464
C06154=1148.682,-114.476,-43.287,178.660,5.955,149.463
C06155=1148.676,-114.226,-43.296,178.662,5.955,149.462
C06156=1148.671,-113.976,-43.305,178.664,5.956,149.462
C06157=1148.665,-113.727,-43.314,178.666,5.957,149.461
C06158=1148.660,-113.477,-43.323,178.668,5.957,149.461
C06159=1148.654,-113.227,-43.332,178.670,5.957,149.461
C06160=1148.649,-112.977,-43.341,178.672,5.957,149.460
C06161=1148.643,-112.728,-43.350,178.674,5.958,149.459
C06162=1148.638,-112.478,-43.359,178.676,5.958,149.459
C06163=1148.633,-112.228,-43.367,178.678,5.958,149.458
C06164=1148.628,-111.978,-43.376,178.680,5.958,149.458
C06165=1148.622,-111.728,-43.385,178.682,5.959,149.457
C06166=1148.617,-111.479,-43.393,178.684,5.960,149.457
C06167=1148.612,-111.229,-43.402,178.686,5.960,149.456
C06168=1148.606,-110.979,-43.411,178.688,5.960,149.456
C06169=1148.601,-110.729,-43.420,178.690,5.960,149.455
C06170=1148.596,-110.479,-43.429,178.692,5.961,149.455
C06171=1148.590,-110.229,-43.438,178.694,5.961,149.454
C06172=1148.584,-109.980,-43.447,178.696,5.962,149.454
C06173=1148.579,-109.730,-43.456,178.698,5.962,149.453
C06174=1148.574,-109.480,-43.464,178.700,5.962,149.453
C06175=1148.569,-109.230,-43.473,178.703,5.963,149.452
C06176=1148.564,-108.981,-43.482,178.704,5.963,149.452
C06177=1148.559,-108.731,-43.491,178.706,5.963,149.451
C06178=1148.553,-108.482,-43.500,178.709,5.964,149.451
C06179=1148.547,-108.231,-43.509,178.710,5.964,149.450
C06180=1148.542,-107.982,-43.518,178.713,5.964,149.449
C06181=1148.537,-107.732,-43.527,178.714,5.964,149.449
C06182=1148.531,-107.482,-43.536,178.717,5.965,149.448
C06183=1148.526,-107.232,-43.545,178.718,5.965,149.448
C06184=1148.521,-106.982,-43.554,178.720,5.966,149.447
C06185=1148.515,-106.733,-43.562,178.723,5.966,149.447
C06186=1148.509,-106.483,-43.572,178.725,5.966,149.446
C06187=1148.504,-106.233,-43.581,178.727,5.967,149.446
C06188=1148.499,-105.983,-43.589,178.728,5.967,149.445
C06189=1148.494,-105.733,-43.598,178.731,5.968,149.445
C06190=1148.489,-105.483,-43.607,178.733,5.968,149.444
C06191=1148.483,-105.233,-43.617,178.735,5.968,149.444
C06192=1148.478,-104.984,-43.626,178.737,5.969,149.443
C06193=1148.473,-104.734,-43.635,178.739,5.969,149.443
C06194=1148.467,-104.485,-43.644,178.741,5.969,149.442
C06195=1148.462,-104.235,-43.653,178.743,5.970,149.442
C06196=1148.456,-103.985,-43.662,178.745,5.970,149.441
C06197=1148.451,-103.735,-43.671,178.747,5.971,149.440
C06198=1148.446,-103.485,-43.680,178.749,5.970,149.440
C06199=1148.440,-103.235,-43.689,178.751,5.971,149.439
C06200=1148.435,-102.964,-43.699,178.754,5.972,149.439
C06201=1148.429,-102.691,-43.710,178.755,5.972,149.438
C06202=1148.422,-102.419,-43.719,178.758,5.972,149.438
C06203=1148.417,-102.148,-43.729,178.760,5.973,149.437
C06204=1148.412,-101.898,-43.738,178.762,5.973,149.437
C06205=1148.406,-101.648,-43.747,178.764,5.973,149.436
C06206=1148.401,-101.398,-43.757,178.766,5.974,149.436
C06207=1148.395,-101.148,-43.766,178.768,5.974,149.435
C06208=1148.391,-100.899,-43.775,178.771,5.975,149.434
C06209=1148.385,-100.649,-43.784,178.773,5.975,149.434
C06210=1148.379,-100.399,-43.794,178.774,5.975,149.433
C06211=1148.374,-100.149,-43.802,178.777,5.976,149.433
C06212=1148.369,-99.899,-43.812,178.779,5.976,149.432
C06213=1148.364,-99.649,-43.822,178.781,5.976,149.432
C06214=1148.358,-99.399,-43.830,178.783,5.977,149.431
C06215=1148.353,-99.150,-43.839,178.785,5.977,149.431
C06216=1148.348,-98.900,-43.850,178.787,5.977,149.430
C06217=1148.342,-98.650,-43.858,178.789,5.978,149.430
C06218=1148.337,-98.400,-43.867,178.791,5.978,149.429
C06219=1148.331,-98.150,-43.877,178.793,5.979,149.429
C06220=1148.326,-97.901,-43.886,178.795,5.979,149.428
C06221=1148.321,-97.652,-43.895,178.798,5.979,149.427
C06222=1148.315,-97.402,-43.904,178.800,5.980,149.427
C06223=1148.310,-97.152,-43.913,178.801,5.980,149.426
C06224=1148.305,-96.903,-43.923,178.804,5.981,149.426
C06225=1148.299,-96.652,-43.932,178.806,5.981,149.425
C06226=1148.294,-96.403,-43.941,178.808,5.981,149.425
C06227=1148.289,-96.153,-43.951,178.810,5.982,149.424
C06228=1148.283,-95.903,-43.960,178.812,5.983,149.424
C06229=1148.278,-95.653,-43.969,178.814,5.983,149.423
C06230=1148.272,-95.404,-43.980,178.816,5.983,149.423
C06231=1148.267,-95.154,-43.988,178.818,5.983,149.422
C06232=1148.262,-94.903,-43.998,178.820,5.984,149.422
C06233=1148.257,-94.654,-44.008,178.822,5.984,149.421
C06234=1148.252,-94.404,-44.017,178.824,5.984,149.420
C06235=1148.246,-94.154,-44.027,178.827,5.985,149.420
C06236=1148.241,-93.905,-44.036,178.829,5.986,149.419
C06237=1148.236,-93.655,-44.045,178.830,5.985,149.419
C06238=1148.230,-93.405,-44.055,178.833,5.986,149.418
C06239=1148.225,-93.155,-44.064,178.835,5.987,149.418
C06240=1148.219,-92.906,-44.074,178.837,5.987,149.417
C06241=1148.214,-92.656,-44.083,178.839,5.987,149.417
C06242=1148.208,-92.406,-44.093,178.842,5.988,149.416
C06243=1148.203,-92.157,-44.102,178.843,5.988,149.416
C06244=1148.198,-91.906,-44.112,178.846,5.988,149.415
C06245=1148.193,-91.657,-44.121,178.848,5.989,149.415
C06246=1148.188,-91.407,-44.130,178.850,5.989,149.414
C06247=1148.182,-91.158,-44.140,178.852,5.990,149.413
C06248=1148.177,-90.908,-44.149,178.854,5.990,149.413
C06249=1148.171,-90.658,-44.159,178.856,5.990,149.413
C06250=1148.166,-90.409,-44.168,178.859,5.991,149.412
C06251=1148.161,-90.158,-44.179,178.861,5.991,149.411
C06252=1148.156,-89.908,-44.188,178.862,5.991,149.411
C06253=1148.150,-89.659,-44.198,178.865,5.992,149.410
C06254=1148.145,-89.409,-44.207,178.867,5.993,149.410
C06255=1148.139,-89.159,-44.217,178.869,5.992,149.409
C06256=1148.134,-88.910,-44.226,178.871,5.993,149.409
C06257=1148.129,-88.660,-44.236,178.873,5.994,149.408
C06258=1148.124,-88.410,-44.245,178.875,5.994,149.407
C06259=1148.118,-88.161,-44.255,178.877,5.994,149.407
C06260=1148.113,-87.911,-44.264,178.880,5.995,149.406
C06261=1148.108,-87.661,-44.275,178.881,5.995,149.406
C06262=1148.102,-87.410,-44.284,178.884,5.995,149.405
C06263=1148.097,-87.161,-44.294,178.886,5.996,149.405
C06264=1148.091,-86.912,-44.304,178.888,5.996,149.404
C06265=1148.086,-86.662,-44.313,178.890,5.997,149.404
C06266=1148.081,-86.412,-44.323,178.893,5.997,149.403
C06267=1148.076,-86.162,-44.332,178.894,5.997,149.403
C06268=1148.071,-85.912,-44.343,178.896,5.998,149.402
C06269=1148.066,-85.663,-44.352,178.899,5.998,149.401
C06270=1148.060,-85.413,-44.362,178.901,5.998,149.401
C06271=1148.054,-85.163,-44.372,178.903,5.999,149.401
C06272=1148.049,-84.913,-44.381,178.905,6.000,149.400
C06273=1148.043,-84.664,-44.391,178.907,6.000,149.399
C06274=1148.039,-84.415,-44.401,178.909,6.000,149.399
C06275=1148.033,-84.164,-44.411,178.911,6.001,149.398
C06276=1148.028,-83.914,-44.421,178.914,6.001,149.398
C06277=1148.023,-83.665,-44.430,178.916,6.001,149.397
C06278=1148.017,-83.415,-44.440,178.918,6.002,149.397
C06279=1148.012,-83.166,-44.450,178.920,6.003,149.396
C06280=1148.007,-82.915,-44.460,178.922,6.003,149.395
C06281=1148.001,-82.665,-44.470,178.924,6.003,149.395
C06282=1147.996,-82.416,-44.479,178.927,6.004,149.395
C06283=1147.991,-82.166,-44.489,178.929,6.004,149.394
C06284=1147.985,-81.917,-44.500,178.931,6.004,149.393
C06285=1147.980,-81.667,-44.509,178.933,6.005,149.393
C06286=1147.975,-81.417,-44.519,178.935,6.006,149.392
C06287=1147.969,-81.167,-44.529,178.937,6.006,149.392
C06288=1147.964,-80.918,-44.539,178.939,6.006,149.391
C06289=1147.959,-80.668,-44.548,178.942,6.007,149.391
C06290=1147.954,-80.418,-44.559,178.944,6.007,149.390
C06291=1147.949,-80.168,-44.569,178.946,6.007,149.389
C06292=1147.943,-79.919,-44.579,178.948,6.008,149.389
C06293=1147.937,-79.669,-44.588,178.951,6.009,149.388
C06294=1147.932,-79.419,-44.598,178.952,6.009,149.388
C06295=1147.927,-79.169,-44.609,178.955,6.009,149.387
C06296=1147.922,-78.920,-44.619,178.957,6.010,149.387
C06297=1147.916,-78.670,-44.629,178.959,6.010,149.386
C06298=1147.911,-78.420,-44.638,178.961,6.010,149.386
C06299=1147.906,-78.170,-44.648,178.963,6.011,149.385
C06300=1147.900,-77.920,-44.659,178.966,6.012,149.384
C06301=1147.895,-77.671,-44.669,178.968,6.012,149.384
C06302=1147.890,-77.422,-44.678,178.970,6.012,149.383
C06303=1147.885,-77.171,-44.688,178.972,6.013,149.383
C06304=1147.879,-76.900,-44.699,178.975,6.013,149.382
C06305=1147.873,-76.629,-44.710,178.977,6.014,149.382
C06306=1147.868,-76.357,-44.721,178.979,6.014,149.381
C06307=1147.861,-76.086,-44.733,178.982,6.014,149.380
C06308=1147.856,-75.836,-44.742,178.984,6.015,149.380
C06309=1147.851,-75.586,-44.752,178.986,6.016,149.379
C06310=1147.845,-75.337,-44.762,178.987,6.016,149.379
C06311=1147.840,-75.087,-44.772,178.990,6.016,149.378
C06312=1147.835,-74.837,-44.783,178.992,6.017,149.378
C06313=1147.829,-74.587,-44.793,178.995,6.018,149.377
C06314=1147.824,-74.338,-44.803,178.997,6.017,149.377
C06315=1147.819,-74.088,-44.813,178.999,6.018,149.376
C06316=1147.814,-73.838,-44.824,179.001,6.019,149.376
C06317=1147.808,-73.589,-44.834,179.004,6.019,149.375
C06318=1147.803,-73.339,-44.844,179.005,6.019,149.374
C06319=1147.798,-73.089,-44.855,179.007,6.020,149.374
C06320=1147.793,-72.840,-44.864,179.010,6.020,149.373
C06321=1147.787,-72.590,-44.874,179.012,6.021,149.373
C06322=1147.782,-72.340,-44.885,179.014,6.021,149.372
C06323=1147.776,-72.090,-44.895,179.017,6.021,149.372
C06324=1147.771,-71.841,-44.905,179.019,6.022,149.371
C06325=1147.766,-71.591,-44.916,179.021,6.023,149.371
C06326=1147.760,-71.341,-44.926,179.023,6.023,149.370
C06327=1147.755,-71.092,-44.936,179.025,6.023,149.369
C06328=1147.750,-70.842,-44.946,179.027,6.024,149.369
C06329=1147.745,-70.592,-44.957,179.030,6.024,149.368
C06330=1147.739,-70.343,-44.967,179.032,6.025,149.368
C06331=1147.734,-70.092,-44.977,179.034,6.025,149.367
C06332=1147.729,-69.843,-44.988,179.037,6.026,149.367
C06333=1147.724,-69.593,-44.998,179.039,6.026,149.366
C06334=1147.718,-69.343,-45.008,179.041,6.027,149.366
C06335=1147.712,-69.093,-45.019,179.043,6.027,149.365
C06336=1147.707,-68.843,-45.029,179.045,6.027,149.364
C06337=1147.702,-68.594,-45.039,179.047,6.028,149.364
C06338=1147.697,-68.344,-45.049,179.050,6.029,149.363
C06339=1147.692,-68.094,-45.060,179.052,6.029,149.363
C06340=1147.686,-67.845,-45.070,179.054,6.029,149.362
C06341=1147.682,-67.595,-45.081,179.057,6.030,149.362
C06342=1147.676,-67.346,-45.091,179.059,6.031,149.361
C06343=1147.670,-67.096,-45.101,179.061,6.031,149.361
C06344=1147.665,-66.846,-45.112,179.063,6.031,149.360
C06345=1147.660,-66.596,-45.122,179.065,6.032,149.359
C06346=1147.655,-66.346,-45.133,179.067,6.032,149.359
C06347=1147.649,-66.096,-45.143,179.070,6.033,149.358
C06348=1147.644,-65.847,-45.154,179.072,6.033,149.358
C06349=1147.639,-65.597,-45.165,179.074,6.034,149.357
C06350=1147.633,-65.348,-45.175,179.076,6.034,149.357
C06351=1147.628,-65.097,-45.185,179.079,6.035,149.356
C06352=1147.623,-64.848,-45.196,179.081,6.036,149.356
C06353=1147.618,-64.598,-45.207,179.083,6.035,149.355
C06354=1147.613,-64.349,-45.217,179.085,6.036,149.354
C06355=1147.607,-64.099,-45.227,179.087,6.037,149.354
C06356=1147.602,-63.849,-45.238,179.090,6.037,149.353
C06357=1147.596,-63.599,-45.248,179.092,6.038,149.353
C06358=1147.592,-63.350,-45.259,179.094,6.038,149.352
C06359=1147.586,-63.100,-45.269,179.096,6.038,149.352
C06360=1147.581,-62.850,-45.280,179.099,6.039,149.351
C06361=1147.575,-62.600,-45.290,179.101,6.040,149.351
C06362=1147.571,-62.351,-45.302,179.103,6.040,149.350
C06363=1147.565,-62.101,-45.312,179.105,6.040,149.349
C06364=1147.560,-61.851,-45.322,179.108,6.041,149.349
C06365=1147.555,-61.602,-45.333,179.110,6.041,149.348
C06366=1147.549,-61.352,-45.344,179.112,6.042,149.348
C06367=1147.544,-61.102,-45.355,179.115,6.042,149.347
C06368=1147.539,-60.852,-45.366,179.116,6.042,149.347
C06369=1147.533,-60.603,-45.376,179.119,6.043,149.346
C06370=1147.528,-60.353,-45.387,179.121,6.044,149.345
C06371=1147.523,-60.104,-45.398,179.123,6.044,149.345
C06372=1147.518,-59.853,-45.408,179.126,6.045,149.344
C06373=1147.512,-59.604,-45.418,179.128,6.046,149.344
C06374=1147.508,-59.354,-45.430,179.130,6.046,149.343
C06375=1147.502,-59.105,-45.440,179.132,6.046,149.343
C06376=1147.496,-58.854,-45.451,179.135,6.047,149.342
C06377=1147.491,-58.605,-45.462,179.137,6.048,149.342
C06378=1147.486,-58.355,-45.473,179.140,6.048,149.341
C06379=1147.481,-58.106,-45.484,179.142,6.049,149.340
C06380=1147.476,-57.856,-45.494,179.143,6.049,149.340
C06381=1147.470,-57.606,-45.504,179.146,6.049,149.339
C06382=1147.465,-57.357,-45.516,179.148,6.050,149.339
C06383=1147.460,-57.107,-45.526,179.150,6.051,149.338
C06384=1147.454,-56.857,-45.538,179.153,6.051,149.338
C06385=1147.449,-56.608,-45.548,179.155,6.051,149.337
C06386=1147.444,-56.358,-45.559,179.157,6.052,149.337
C06387=1147.439,-56.108,-45.570,179.160,6.052,149.336
C06388=1147.434,-55.858,-45.580,179.162,6.053,149.335
C06389=1147.428,-55.608,-45.592,179.164,6.053,149.335
C06390=1147.423,-55.359,-45.602,179.167,6.054,149.334
C06391=1147.418,-55.109,-45.613,179.169,6.055,149.334
C06392=1147.412,-54.860,-45.624,179.171,6.054,149.333
C06393=1147.408,-54.610,-45.635,179.173,6.055,149.333
C06394=1147.402,-54.359,-45.646,179.175,6.056,149.332
C06395=1147.397,-54.110,-45.657,179.178,6.056,149.331
C06396=1147.392,-53.860,-45.668,179.180,6.057,149.331
C06397=1147.386,-53.611,-45.678,179.183,6.058,149.330
C06398=1147.382,-53.362,-45.690,179.184,6.058,149.330
C06399=1147.376,-53.111,-45.701,179.187,6.058,149.329
C06400=1147.371,-52.862,-45.712,179.189,6.059,149.329
C06401=1147.366,-52.612,-45.722,179.191,6.060,149.328
C06402=1147.360,-52.363,-45.733,179.194,6.060,149.328
C06403=1147.354,-52.112,-45.745,179.196,6.061,149.327
C06404=1147.350,-51.863,-45.756,179.198,6.062,149.326
C06405=1147.344,-51.614,-45.767,179.200,6.061,149.326
C06406=1147.339,-51.363,-45.778,179.203,6.062,149.325
C06407=1147.334,-51.114,-45.789,179.205,6.063,149.325
C06408=1147.328,-50.843,-45.801,179.208,6.063,149.324
C06409=1147.323,-50.573,-45.813,179.210,6.063,149.323
C06410=1147.317,-50.302,-45.825,179.212,6.064,149.323
C06411=1147.311,-50.032,-45.837,179.215,6.065,149.322
C06412=1147.306,-49.781,-45.847,179.217,6.065,149.322
C06413=1147.300,-49.532,-45.859,179.219,6.066,149.321
C06414=1147.295,-49.282,-45.870,179.222,6.067,149.320
C06415=1147.290,-49.032,-45.881,179.224,6.067,149.320
C06416=1147.284,-48.783,-45.892,179.227,6.068,149.319
C06417=1147.280,-48.533,-45.904,179.229,6.069,149.319
C06418=1147.275,-48.283,-45.914,179.231,6.069,149.318
C06419=1147.269,-48.034,-45.926,179.233,6.069,149.318
C06420=1147.264,-47.784,-45.937,179.236,6.070,149.317
C06421=1147.259,-47.534,-45.949,179.238,6.070,149.316
C06422=1147.253,-47.285,-45.959,179.240,6.071,149.316
C06423=1147.248,-47.035,-45.970,179.243,6.072,149.315
C06424=1147.243,-46.785,-45.982,179.245,6.072,149.315
C06425=1147.237,-46.536,-45.992,179.247,6.073,149.314
C06426=1147.232,-46.286,-46.004,179.250,6.073,149.314
C06427=1147.227,-46.036,-46.016,179.252,6.073,149.313
C06428=1147.222,-45.786,-46.027,179.254,6.074,149.313
C06429=1147.216,-45.537,-46.038,179.257,6.074,149.312
C06430=1147.211,-45.287,-46.049,179.259,6.075,149.311
C06431=1147.206,-45.037,-46.061,179.261,6.076,149.311
C06432=1147.201,-44.788,-46.072,179.264,6.076,149.310
C06433=1147.196,-44.538,-46.083,179.266,6.077,149.310
C06434=1147.190,-44.288,-46.094,179.268,6.078,149.309
C06435=1147.186,-44.038,-46.106,179.271,6.078,149.309
C06436=1147.180,-43.789,-46.117,179.273,6.079,149.308
C06437=1147.175,-43.539,-46.128,179.275,6.079,149.307
C06438=1147.169,-43.289,-46.140,179.277,6.080,149.307
C06439=1147.165,-43.040,-46.152,179.280,6.080,149.306
C06440=1147.159,-42.791,-46.163,179.282,6.081,149.306
C06441=1147.154,-42.540,-46.174,179.284,6.082,149.305
C06442=1147.148,-42.290,-46.186,179.287,6.082,149.305
C06443=1147.144,-42.041,-46.197,179.289,6.083,149.304
C06444=1147.138,-41.792,-46.208,179.292,6.083,149.303
C06445=1147.133,-41.542,-46.220,179.294,6.084,149.303
C06446=1147.127,-41.292,-46.232,179.296,6.085,149.302
C06447=1147.123,-41.042,-46.243,179.299,6.085,149.302
C06448=1147.117,-40.792,-46.255,179.301,6.086,149.301
C06449=1147.112,-40.544,-46.266,179.303,6.086,149.301
C06450=1147.107,-40.294,-46.278,179.305,6.086,149.300
C06451=1147.102,-40.043,-46.288,179.307,6.087,149.300
C06452=1147.096,-39.793,-46.300,179.310,6.088,149.299
C06453=1147.091,-39.544,-46.311,179.312,6.088,149.298
C06454=1147.085,-39.295,-46.323,179.315,6.089,149.298
C06455=1147.081,-39.045,-46.334,179.317,6.090,149.297
C06456=1147.075,-38.795,-46.346,179.320,6.090,149.297
C06457=1147.070,-38.545,-46.358,179.322,6.091,149.296
C06458=1147.065,-38.296,-46.369,179.324,6.091,149.296
C06459=1147.059,-38.046,-46.381,179.327,6.092,149.295
C06460=1147.054,-37.797,-46.392,179.329,6.093,149.294
C06461=1147.049,-37.547,-46.404,179.332,6.093,149.294
C06462=1147.044,-37.297,-46.416,179.334,6.094,149.293
C06463=1147.039,-37.047,-46.427,179.336,6.095,149.293
C06464=1147.033,-36.798,-46.439,179.339,6.095,149.292
C06465=1147.028,-36.548,-46.450,179.340,6.095,149.292
C06466=1147.023,-36.299,-46.462,179.343,6.095,149.291
C06467=1147.018,-36.049,-46.474,179.345,6.096,149.290
C06468=1147.013,-35.799,-46.486,179.347,6.097,149.290
C06469=1147.007,-35.549,-46.497,179.350,6.097,149.289
C06470=1147.002,-35.299,-46.509,179.352,6.098,149.289
C06471=1146.997,-35.051,-46.520,179.355,6.099,149.288
C06472=1146.991,-34.801,-46.532,179.357,6.099,149.288
C06473=1146.986,-34.551,-46.544,179.359,6.100,149.287
C06474=1146.981,-34.301,-46.555,179.362,6.101,149.286
C06475=1146.976,-34.051,-46.567,179.364,6.101,149.286
C06476=1146.971,-33.802,-46.580,179.367,6.102,149.285
C06477=1146.966,-33.552,-46.591,179.369,6.103,149.285
C06478=1146.961,-33.302,-46.603,179.371,6.103,149.284
C06479=1146.955,-33.053,-46.615,179.374,6.104,149.284
C06480=1146.950,-32.803,-46.626,179.376,6.105,149.283
C06481=1146.944,-32.553,-46.638,179.379,6.105,149.282
C06482=1146.939,-32.304,-46.650,179.381,6.106,149.282
C06483=1146.935,-32.054,-46.662,179.383,6.106,149.281
C06484=1146.929,-31.805,-46.673,179.386,6.107,149.281
C06485=1146.924,-31.555,-46.685,179.388,6.108,149.280
C06486=1146.918,-31.305,-46.697,179.390,6.108,149.280
C06487=1146.914,-31.056,-46.709,179.393,6.109,149.279
C06488=1146.908,-30.806,-46.721,179.395,6.109,149.279
C06489=1146.903,-30.556,-46.733,179.397,6.110,149.278
C06490=1146.898,-30.306,-46.745,179.400,6.111,149.277
C06491=1146.893,-30.057,-46.757,179.402,6.111,149.277
C06492=1146.887,-29.808,-46.768,179.404,6.112,149.276
C06493=1146.882,-29.558,-46.780,179.407,6.113,149.276
C06494=1146.876,-29.308,-46.792,179.409,6.113,149.275
C06495=1146.872,-29.059,-46.804,179.412,6.114,149.275
C06496=1146.867,-28.809,-46.816,179.414,6.115,149.274
C06497=1146.861,-28.559,-46.828,179.416,6.115,149.274
C06498=1146.856,-28.310,-46.841,179.419,6.116,149.273
C06499=1146.851,-28.060,-46.852,179.421,6.117,149.272
C06500=1146.846,-27.810,-46.864,179.424,6.117,149.272
C06501=1146.841,-27.561,-46.876,179.426,6.118,149.271
C06502=1146.835,-27.311,-46.888,179.429,6.118,149.271
C06503=1146.830,-27.061,-46.900,179.431,6.119,149.270
C06504=1146.825,-26.811,-46.913,179.433,6.120,149.270
C06505=1146.820,-26.562,-46.924,179.436,6.120,149.269
C06506=1146.815,-26.312,-46.936,179.438,6.121,149.268
C06507=1146.810,-26.063,-46.949,179.441,6.121,149.268
C06508=1146.804,-25.813,-46.960,179.443,6.122,149.267
C06509=1146.799,-25.563,-46.973,179.445,6.123,149.267
C06510=1146.794,-25.313,-46.985,179.448,6.123,149.266
C06511=1146.788,-25.063,-46.997,179.450,6.124,149.266
C06512=1146.783,-24.794,-47.010,179.452,6.125,149.265
C06513=1146.778,-24.523,-47.023,179.455,6.125,149.264
C06514=1146.772,-24.254,-47.036,179.457,6.126,149.264
C06515=1146.767,-23.983,-47.049,179.460,6.126,149.263
C06516=1146.761,-23.734,-47.062,179.462,6.127,149.263
C06517=1146.756,-23.484,-47.073,179.465,6.128,149.262
C06518=1146.751,-23.235,-47.086,179.467,6.128,149.261
C06519=1146.745,-22.985,-47.098,179.470,6.129,149.261
C06520=1146.740,-22.736,-47.111,179.472,6.130,149.260
C06521=1146.735,-22.486,-47.122,179.474,6.130,149.260
C06522=1146.730,-22.236,-47.135,179.477,6.132,149.259
C06523=1146.724,-21.986,-47.147,179.479,6.132,149.259
C06524=1146.719,-21.737,-47.160,179.482,6.133,149.258
C06525=1146.714,-21.487,-47.171,179.484,6.134,149.257
C06526=1146.709,-21.238,-47.184,179.487,6.134,149.257
C06527=1146.704,-20.988,-47.197,179.489,6.135,149.256
C06528=1146.699,-20.738,-47.209,179.491,6.136,149.256
C06529=1146.694,-20.488,-47.221,179.494,6.136,149.255
C06530=1146.688,-20.239,-47.233,179.496,6.137,149.255
C06531=1146.683,-19.989,-47.246,179.499,6.137,149.254
C06532=1146.678,-19.739,-47.258,179.501,6.138,149.253
C06533=1146.672,-19.490,-47.270,179.504,6.138,149.253
C06534=1146.667,-19.241,-47.283,179.506,6.139,149.252
C06535=1146.662,-18.991,-47.295,179.508,6.140,149.252
C06536=1146.657,-18.741,-47.308,179.511,6.140,149.251
C06537=1146.651,-18.491,-47.319,179.513,6.141,149.251
C06538=1146.647,-18.241,-47.332,179.516,6.142,149.250
C06539=1146.642,-17.992,-47.345,179.518,6.142,149.250
C06540=1146.636,-17.742,-47.357,179.520,6.143,149.249
C06541=1146.631,-17.493,-47.369,179.523,6.144,149.248
C06542=1146.626,-17.244,-47.382,179.525,6.144,149.248
C06543=1146.621,-16.994,-47.394,179.528,6.146,149.247
C06544=1146.616,-16.744,-47.407,179.530,6.146,149.247
C06545=1146.611,-16.494,-47.420,179.533,6.147,149.246
C06546=1146.606,-16.244,-47.431,179.535,6.148,149.246
C06547=1146.600,-15.995,-47.444,179.538,6.148,149.245
C06548=1146.595,-15.746,-47.457,179.540,6.149,149.244
C06549=1146.589,-15.496,-47.470,179.542,6.150,149.244
C06550=1146.584,-15.246,-47.482,179.545,6.150,149.243
C06551=1146.579,-14.996,-47.495,179.547,6.151,149.243
C06552=1146.574,-14.747,-47.507,179.550,6.151,149.242
C06553=1146.569,-14.498,-47.520,179.552,6.152,149.242
C06554=1146.564,-14.248,-47.532,179.554,6.153,149.241
C06555=1146.559,-13.998,-47.544,179.557,6.153,149.240
C06556=1146.554,-13.748,-47.557,179.559,6.154,149.240
C06557=1146.548,-13.499,-47.571,179.562,6.155,149.239
C06558=1146.543,-13.249,-47.583,179.564,6.156,149.239
C06559=1146.538,-12.999,-47.595,179.567,6.157,149.238
C06560=1146.533,-12.750,-47.608,179.569,6.157,149.238
C06561=1146.528,-12.500,-47.621,179.572,6.158,149.237
C06562=1146.523,-12.251,-47.633,179.574,6.159,149.236
C06563=1146.518,-12.001,-47.646,179.576,6.159,149.236
C06564=1146.512,-11.752,-47.659,179.579,6.160,149.235
C06565=1146.507,-11.502,-47.671,179.581,6.161,149.235
C06566=1146.502,-11.252,-47.684,179.583,6.161,149.234
C06567=1146.497,-11.002,-47.696,179.586,6.162,149.234
C06568=1146.492,-10.753,-47.709,179.589,6.163,149.233
C06569=1146.486,-10.504,-47.722,179.591,6.164,149.233
C06570=1146.481,-10.254,-47.735,179.594,6.164,149.232
C06571=1146.476,-10.004,-47.748,179.596,6.165,149.231
C06572=1146.471,-9.755,-47.760,179.598,6.166,149.231
C06573=1146.467,-9.505,-47.773,179.601,6.166,149.230
C06574=1146.461,-9.255,-47.787,179.603,6.167,149.230
C06575=1146.456,-9.006,-47.799,179.606,6.168,149.229
C06576=1146.451,-8.757,-47.812,179.608,6.168,149.229
C06577=1146.446,-8.506,-47.824,179.611,6.170,149.228
C06578=1146.440,-8.256,-47.837,179.613,6.171,149.227
C06579=1146.435,-8.007,-47.850,179.616,6.171,149.227
C06580=1146.430,-7.757,-47.863,179.618,6.172,149.226
C06581=1146.424,-7.507,-47.876,179.620,6.173,149.226
C06582=1146.419,-7.258,-47.889,179.623,6.173,149.225
C06583=1146.414,-7.009,-47.901,179.625,6.174,149.225
C06584=1146.410,-6.759,-47.914,179.628,6.174,149.224
C06585=1146.404,-6.510,-47.928,179.631,6.176,149.223
C06586=1146.399,-6.260,-47.941,179.633,6.176,149.223
C06587=1146.394,-6.010,-47.954,179.635,6.177,149.222
C06588=1146.388,-5.761,-47.967,179.638,6.178,149.222
C06589=1146.383,-5.511,-47.979,179.640,6.178,149.221
C06590=1146.379,-5.261,-47.992,179.642,6.179,149.221
C06591=1146.373,-5.012,-48.006,179.645,6.180,149.220
C06592=1146.368,-4.762,-48.018,179.647,6.180,149.220
C06593=1146.363,-4.512,-48.031,179.650,6.182,149.219
C06594=1146.357,-4.263,-48.044,179.653,6.182,149.218
C06595=1146.352,-4.013,-48.057,179.655,6.183,149.218
C06596=1146.348,-3.763,-48.070,179.657,6.184,149.217
C06597=1146.342,-3.514,-48.084,179.660,6.184,149.217
C06598=1146.337,-3.265,-48.096,179.662,6.185,149.216
C06599=1146.332,-3.015,-48.110,179.664,6.186,149.216
C06600=1146.327,-2.766,-48.123,179.668,6.187,149.215
C06601=1146.322,-2.515,-48.136,179.670,6.188,149.214
C06602=1146.316,-2.266,-48.149,179.673,6.188,149.214
C06603=1146.311,-2.017,-48.161,179.675,6.189,149.213
C06604=1146.306,-1.767,-48.176,179.677,6.190,149.213
C06605=1146.301,-1.518,-48.188,179.680,6.190,149.212
C06606=1146.295,-1.268,-48.201,179.682,6.192,149.212
C06607=1146.291,-1.018,-48.214,179.685,6.192,149.211
C06608=1146.286,-0.769,-48.228,179.687,6.193,149.211
C06609=1146.281,-0.519,-48.241,179.690,6.193,149.210
C06610=1146.276,-0.270,-48.254,179.692,6.194,149.209
C06611=1146.270,-0.019,-48.267,179.694,6.195,149.209
C06612=1146.266,0.230,-48.281,179.697,6.196,149.208
C06613=1146.260,0.479,-48.294,179.700,6.197,149.208
C06614=1146.255,0.729,-48.307,179.702,6.198,149.207
C06615=1146.249,0.979,-48.320,179.704,6.198,149.207
C06616=1146.245,1.248,-48.334,179.707,6.199,149.206
C06617=1146.239,1.518,-48.349,179.710,6.200,149.205
C06618=1146.233,1.787,-48.363,179.713,6.201,149.205
C06619=1146.227,2.057,-48.378,179.715,6.201,149.204
C06620=1146.222,2.305,-48.391,179.718,6.203,149.204
C06621=1146.217,2.556,-48.405,179.721,6.203,149.203
C06622=1146.212,2.805,-48.417,179.723,6.204,149.202
C06623=1146.207,3.055,-48.431,179.725,6.205,149.202
C06624=1146.202,3.304,-48.444,179.728,6.205,149.201
C06625=1146.197,3.554,-48.458,179.730,6.207,149.201
C06626=1146.192,3.803,-48.471,179.733,6.207,149.200
C06627=1146.186,4.053,-48.484,179.735,6.208,149.200
C06628=1146.182,4.302,-48.498,179.738,6.209,149.199
C06629=1146.176,4.552,-48.511,179.740,6.210,149.199
C06630=1146.170,4.802,-48.525,179.743,6.211,149.198
C06631=1146.166,5.051,-48.538,179.745,6.212,149.197
C06632=1146.160,5.301,-48.551,179.748,6.212,149.197
C06633=1146.156,5.550,-48.565,179.750,6.213,149.196
C06634=1146.150,5.800,-48.578,179.752,6.214,149.196
C06635=1146.145,6.050,-48.593,179.756,6.215,149.195
C06636=1146.140,6.299,-48.605,179.758,6.216,149.195
C06637=1146.135,6.549,-48.619,179.761,6.216,149.194
C06638=1146.130,6.798,-48.632,179.763,6.217,149.193
C06639=1146.125,7.048,-48.646,179.765,6.218,149.193
C06640=1146.119,7.298,-48.660,179.768,6.219,149.192
C06641=1146.115,7.547,-48.673,179.770,6.220,149.192
C06642=1146.110,7.797,-48.687,179.773,6.220,149.191
C06643=1146.104,8.046,-48.701,179.775,6.221,149.191
C06644=1146.100,8.296,-48.714,179.778,6.222,149.190
C06645=1146.094,8.545,-48.728,179.781,6.223,149.190
C06646=1146.089,8.796,-48.741,179.783,6.224,149.189
C06647=1146.084,9.044,-48.754,179.785,6.224,149.188
C06648=1146.079,9.295,-48.768,179.788,6.225,149.188
C06649=1146.073,9.544,-48.782,179.791,6.226,149.187
C06650=1146.069,9.793,-48.796,179.793,6.227,149.187
C06651=1146.064,10.043,-48.809,179.796,6.228,149.186
C06652=1146.058,10.292,-48.823,179.798,6.228,149.186
C06653=1146.053,10.543,-48.837,179.801,6.230,149.185
C06654=1146.048,10.791,-48.850,179.803,6.231,149.185
C06655=1146.043,11.041,-48.864,179.805,6.231,149.184
C06656=1146.038,11.291,-48.878,179.808,6.232,149.183
C06657=1146.032,11.540,-48.892,179.811,6.233,149.183
C06658=1146.028,11.790,-48.905,179.813,6.234,149.182
C06659=1146.022,12.039,-48.919,179.816,6.235,149.182
C06660=1146.017,12.289,-48.933,179.818,6.236,149.181
C06661=1146.012,12.539,-48.947,179.821,6.237,149.181
C06662=1146.007,12.788,-48.960,179.823,6.238,149.180
C06663=1146.002,13.038,-48.974,179.826,6.238,149.179
C06664=1145.997,13.288,-48.988,179.828,6.239,149.179
C06665=1145.992,13.537,-49.002,179.831,6.240,149.178
C06666=1145.987,13.787,-49.016,179.833,6.241,149.178
C06667=1145.982,14.036,-49.029,179.836,6.242,149.177
C06668=1145.977,14.285,-49.043,179.838,6.242,149.177
C06669=1145.972,14.536,-49.057,179.841,6.244,149.176
C06670=1145.966,14.785,-49.071,179.844,6.244,149.176
C06671=1145.961,15.034,-49.085,179.846,6.245,149.175
C06672=1145.957,15.284,-49.099,179.849,6.245,149.174
C06673=1145.951,15.533,-49.113,179.851,6.247,149.174
C06674=1145.946,15.783,-49.126,179.853,6.248,149.174
C06675=1145.941,16.033,-49.141,179.856,6.248,149.173
C06676=1145.936,16.282,-49.154,179.858,6.249,149.172
C06677=1145.931,16.532,-49.169,179.862,6.250,149.172
C06678=1145.926,16.781,-49.183,179.864,6.251,149.171
C06679=1145.921,17.031,-49.197,179.866,6.252,149.171
C06680=1145.916,17.280,-49.210,179.869,6.253,149.170
C06681=1145.911,17.530,-49.224,179.871,6.254,149.170
C06682=1145.906,17.780,-49.238,179.874,6.255,149.169
C06683=1145.900,18.029,-49.252,179.876,6.255,149.169
C06684=1145.895,18.279,-49.267,179.879,6.257,149.168
C06685=1145.890,18.528,-49.281,179.882,6.257,149.167
C06686=1145.885,18.778,-49.295,179.884,6.258,149.167
C06687=1145.880,19.027,-49.309,179.887,6.260,149.166
C06688=1145.875,19.277,-49.323,179.889,6.260,149.166
C06689=1145.870,19.526,-49.338,179.892,6.261,149.165
C06690=1145.865,19.777,-49.351,179.894,6.262,149.165
C06691=1145.859,20.026,-49.365,179.897,6.263,149.164
C06692=1145.854,20.275,-49.379,179.899,6.264,149.163
C06693=1145.849,20.525,-49.394,179.902,6.265,149.163
C06694=1145.844,20.775,-49.408,179.905,6.266,149.162
C06695=1145.839,21.024,-49.422,179.907,6.267,149.162
C06696=1145.834,21.273,-49.436,179.910,6.267,149.161
C06697=1145.829,21.523,-49.450,179.912,6.269,149.161
C06698=1145.824,21.773,-49.464,179.915,6.269,149.160
C06699=1145.819,22.022,-49.478,179.917,6.270,149.160
C06700=1145.813,22.272,-49.493,179.919,6.271,149.159
C06701=1145.808,22.521,-49.507,179.923,6.272,149.158
C06702=1145.804,22.770,-49.522,179.925,6.273,149.158
C06703=1145.799,23.020,-49.536,179.927,6.273,149.157
C06704=1145.793,23.269,-49.550,179.930,6.275,149.157
C06705=1145.788,23.519,-49.565,179.933,6.275,149.156
C06706=1145.783,23.769,-49.579,179.935,6.276,149.156
C06707=1145.778,24.018,-49.593,179.938,6.278,149.155
C06708=1145.773,24.268,-49.607,179.940,6.278,149.155
C06709=1145.768,24.517,-49.621,179.943,6.279,149.154
C06710=1145.763,24.767,-49.636,179.946,6.280,149.153
C06711=1145.758,25.016,-49.650,179.948,6.281,149.153
C06712=1145.753,25.266,-49.665,179.950,6.282,149.153
C06713=1145.748,25.515,-49.679,179.953,6.283,149.152
C06714=1145.743,25.765,-49.693,179.956,6.284,149.151
C06715=1145.738,26.014,-49.707,179.958,6.285,149.151
C06716=1145.732,26.264,-49.722,179.961,6.286,149.150
C06717=1145.727,26.514,-49.736,179.963,6.287,149.150
C06718=1145.722,26.763,-49.751,179.966,6.287,149.149
C06719=1145.717,27.013,-49.766,179.969,6.289,149.149
C06720=1145.712,27.281,-49.781,179.971,6.290,149.148
C06721=1145.706,27.551,-49.797,179.974,6.291,149.147
C06722=1145.701,27.820,-49.813,179.977,6.292,149.147
C06723=1145.695,28.088,-49.828,179.980,6.293,149.146
C06724=1145.690,28.338,-49.842,179.982,6.294,149.146
C06725=1145.685,28.587,-49.857,179.985,6.295,149.145
C06726=1145.680,28.837,-49.872,179.987,6.296,149.145
C06727=1145.675,29.086,-49.887,179.990,6.297,149.144
C06728=1145.670,29.336,-49.901,179.993,6.298,149.144
C06729=1145.665,29.586,-49.915,179.995,6.299,149.143
C06730=1145.660,29.835,-49.930,179.998,6.299,149.142
C06731=1145.655,30.085,-49.945,-180.000,6.301,149.142
C06732=1145.650,30.335,-49.959,-179.997,6.302,149.141
C06733=1145.645,30.584,-49.974,-179.995,6.302,149.141
C06734=1145.640,30.833,-49.988,-179.992,6.304,149.140
C06735=1145.635,31.083,-50.002,-179.989,6.304,149.140
C06736=1145.629,31.332,-50.018,-179.987,6.306,149.139
C06737=1145.624,31.582,-50.032,-179.984,6.307,149.139
C06738=1145.620,31.831,-50.047,-179.982,6.307,149.138
C06739=1145.614,32.081,-50.062,-179.979,6.309,149.138
C06740=1145.609,32.330,-50.076,-179.976,6.309,149.137
C06741=1145.604,32.580,-50.091,-179.974,6.310,149.137
C06742=1145.599,32.829,-50.106,-179.971,6.312,149.136
C06743=1145.594,33.079,-50.121,-179.969,6.312,149.135
C06744=1145.589,33.328,-50.136,-179.966,6.314,149.135
C06745=1145.584,33.577,-50.151,-179.963,6.314,149.134
C06746=1145.579,33.827,-50.165,-179.961,6.315,149.134
C06747=1145.574,34.077,-50.180,-179.958,6.317,149.133
C06748=1145.569,34.326,-50.195,-179.956,6.317,149.133
C06749=1145.563,34.576,-50.210,-179.953,6.319,149.132
C06750=1145.559,34.825,-50.225,-179.950,6.319,149.132
C06751=1145.554,35.075,-50.239,-179.948,6.320,149.131
C06752=1145.548,35.325,-50.254,-179.945,6.322,149.131
C06753=1145.543,35.574,-50.269,-179.943,6.322,149.130
C06754=1145.539,35.823,-50.284,-179.940,6.324,149.130
C06755=1145.533,36.073,-50.299,-179.937,6.324,149.129
C06756=1145.528,36.322,-50.314,-179.935,6.325,149.128
C06757=1145.524,36.572,-50.329,-179.933,6.327,149.128
C06758=1145.518,36.822,-50.343,-179.930,6.327,149.127
C06759=1145.513,37.071,-50.358,-179.927,6.329,149.127
C06760=1145.508,37.321,-50.373,-179.924,6.329,149.126
C06761=1145.503,37.570,-50.388,-179.922,6.330,149.126
C06762=1145.498,37.819,-50.404,-179.920,6.332,149.125
C06763=1145.493,38.069,-50.418,-179.917,6.332,149.125
C06764=1145.488,38.318,-50.433,-179.914,6.334,149.124
C06765=1145.482,38.568,-50.448,-179.911,6.334,149.123
C06766=1145.478,38.818,-50.463,-179.909,6.336,149.123
C06767=1145.473,39.067,-50.479,-179.907,6.337,149.123
C06768=1145.468,39.317,-50.493,-179.904,6.337,149.122
C06769=1145.463,39.566,-50.509,-179.901,6.339,149.121
C06770=1145.458,39.815,-50.524,-179.899,6.339,149.121
C06771=1145.453,40.065,-50.539,-179.896,6.341,149.120
C06772=1145.448,40.314,-50.554,-179.894,6.342,149.120
C06773=1145.442,40.564,-50.569,-179.890,6.343,149.119
C06774=1145.438,40.813,-50.584,-179.888,6.344,149.119
C06775=1145.432,41.063,-50.599,-179.886,6.345,149.118
C06776=1145.427,41.312,-50.614,-179.883,6.346,149.118
C06777=1145.423,41.562,-50.630,-179.881,6.347,149.117
C06778=1145.418,41.811,-50.645,-179.877,6.348,149.117
C06779=1145.412,42.061,-50.660,-179.875,6.349,149.116
C06780=1145.408,42.310,-50.675,-179.872,6.351,149.116
C06781=1145.402,42.560,-50.691,-179.870,6.351,149.115
C06782=1145.397,42.809,-50.705,-179.867,6.353,149.114
C06783=1145.392,43.058,-50.721,-179.864,6.353,149.114
C06784=1145.387,43.308,-50.735,-179.862,6.355,149.113
C06785=1145.382,43.558,-50.751,-179.860,6.356,149.113
C06786=1145.377,43.808,-50.767,-179.857,6.356,149.112
C06787=1145.372,44.057,-50.782,-179.854,6.358,149.112
C06788=1145.367,44.306,-50.797,-179.852,6.359,149.111
C06789=1145.362,44.555,-50.812,-179.849,6.360,149.111
C06790=1145.357,44.805,-50.827,-179.847,6.361,149.110
C06791=1145.352,45.055,-50.843,-179.843,6.362,149.110
C06792=1145.347,45.304,-50.858,-179.841,6.363,149.109
C06793=1145.342,45.554,-50.874,-179.838,6.364,149.109
C06794=1145.337,45.803,-50.889,-179.836,6.365,149.108
C06795=1145.332,46.052,-50.904,-179.833,6.367,149.108
C06796=1145.327,46.302,-50.920,-179.831,6.367,149.107
C06797=1145.322,46.551,-50.935,-179.828,6.369,149.106
C06798=1145.317,46.801,-50.951,-179.825,6.369,149.106
C06799=1145.312,47.050,-50.967,-179.822,6.371,149.105
C06800=1145.307,47.299,-50.982,-179.820,6.372,149.105
C06801=1145.302,47.549,-50.998,-179.817,6.373,149.104
C06802=1145.297,47.799,-51.013,-179.815,6.374,149.104
C06803=1145.292,48.048,-51.028,-179.813,6.375,149.103
C06804=1145.287,48.297,-51.044,-179.810,6.376,149.103
C06805=1145.282,48.547,-51.060,-179.807,6.377,149.102
C06806=1145.277,48.796,-51.075,-179.804,6.378,149.102
C06807=1145.272,49.046,-51.090,-179.802,6.379,149.101
C06808=1145.266,49.295,-51.106,-179.799,6.380,149.101
C06809=1145.262,49.545,-51.122,-179.797,6.381,149.100
C06810=1145.257,49.794,-51.137,-179.794,6.383,149.100
C06811=1145.252,50.044,-51.152,-179.791,6.383,149.099
C06812=1145.247,50.294,-51.168,-179.789,6.385,149.099
C06813=1145.242,50.543,-51.183,-179.786,6.386,149.098
C06814=1145.237,50.792,-51.199,-179.783,6.387,149.098
C06815=1145.231,51.042,-51.214,-179.781,6.388,149.097
C06816=1145.227,51.291,-51.231,-179.778,6.389,149.096
C06817=1145.222,51.540,-51.246,-179.775,6.391,149.096
C06818=1145.217,51.790,-51.262,-179.772,6.391,149.095
C06819=1145.212,52.040,-51.278,-179.770,6.393,149.095
C06820=1145.207,52.289,-51.293,-179.768,6.394,149.094
C06821=1145.201,52.539,-51.309,-179.764,6.395,149.094
C06822=1145.196,52.788,-51.324,-179.762,6.396,149.093
C06823=1145.192,53.037,-51.341,-179.759,6.398,149.093
C06824=1145.187,53.306,-51.358,-179.757,6.398,149.092
C06825=1145.181,53.574,-51.375,-179.754,6.400,149.092
C06826=1145.175,53.843,-51.391,-179.751,6.401,149.091
C06827=1145.170,54.113,-51.408,-179.748,6.402,149.090
C06828=1145.165,54.361,-51.425,-179.745,6.403,149.090
C06829=1145.160,54.611,-51.440,-179.743,6.405,149.090
C06830=1145.155,54.861,-51.456,-179.740,6.405,149.089
C06831=1145.150,55.110,-51.471,-179.737,6.407,149.088
C06832=1145.145,55.359,-51.487,-179.735,6.408,149.088
C06833=1145.141,55.609,-51.503,-179.732,6.409,149.087
C06834=1145.135,55.858,-51.519,-179.730,6.410,149.087
C06835=1145.130,56.107,-51.535,-179.727,6.412,149.086
C06836=1145.125,56.357,-51.551,-179.724,6.412,149.086
C06837=1145.120,56.607,-51.567,-179.722,6.414,149.085
C06838=1145.115,56.856,-51.583,-179.719,6.415,149.085
C06839=1145.110,57.105,-51.599,-179.716,6.416,149.084
C06840=1145.105,57.355,-51.615,-179.713,6.417,149.084
C06841=1145.100,57.604,-51.631,-179.711,6.418,149.083
C06842=1145.095,57.854,-51.647,-179.708,6.420,149.083
C06843=1145.090,58.104,-51.663,-179.706,6.420,149.082
C06844=1145.085,58.353,-51.679,-179.703,6.422,149.082
C06845=1145.080,58.602,-51.694,-179.700,6.423,149.081
C06846=1145.076,58.851,-51.711,-179.698,6.424,149.081
C06847=1145.070,59.101,-51.726,-179.696,6.425,149.080
C06848=1145.066,59.350,-51.743,-179.692,6.426,149.080
C06849=1145.061,59.599,-51.759,-179.690,6.428,149.079
C06850=1145.056,59.850,-51.775,-179.687,6.429,149.079
C06851=1145.051,60.098,-51.791,-179.684,6.430,149.078
C06852=1145.045,60.348,-51.806,-179.682,6.431,149.078
C06853=1145.040,60.598,-51.824,-179.679,6.433,149.077
C06854=1145.035,60.847,-51.839,-179.677,6.433,149.077
C06855=1145.030,61.096,-51.856,-179.674,6.435,149.076
C06856=1145.025,61.346,-51.872,-179.671,6.436,149.076
C06857=1145.020,61.595,-51.888,-179.669,6.437,149.075
C06858=1145.015,61.845,-51.904,-179.666,6.439,149.075
C06859=1145.010,62.094,-51.921,-179.664,6.439,149.074
C06860=1145.005,62.343,-51.937,-179.660,6.441,149.073
C06861=1145.001,62.593,-51.953,-179.658,6.442,149.073
C06862=1144.995,62.842,-51.969,-179.656,6.443,149.073
C06863=1144.991,63.092,-51.985,-179.652,6.444,149.072
C06864=1144.986,63.341,-52.001,-179.650,6.445,149.072
C06865=1144.981,63.591,-52.017,-179.647,6.447,149.071
C06866=1144.976,63.840,-52.034,-179.644,6.448,149.070
C06867=1144.971,64.089,-52.051,-179.642,6.449,149.070
C06868=1144.965,64.339,-52.066,-179.639,6.451,149.070
C06869=1144.961,64.588,-52.083,-179.637,6.451,149.069
C06870=1144.956,64.837,-52.099,-179.634,6.453,149.068
C06871=1144.951,65.087,-52.115,-179.631,6.455,149.068
C06872=1144.946,65.336,-52.132,-179.628,6.455,149.067
C06873=1144.941,65.585,-52.148,-179.626,6.457,149.067
C06874=1144.936,65.836,-52.165,-179.624,6.458,149.066
C06875=1144.931,66.085,-52.181,-179.620,6.459,149.066
C06876=1144.926,66.334,-52.198,-179.618,6.461,149.065
C06877=1144.921,66.584,-52.213,-179.615,6.461,149.065
C06878=1144.916,66.833,-52.230,-179.612,6.463,149.064
C06879=1144.911,67.082,-52.246,-179.609,6.464,149.064
C06880=1144.906,67.332,-52.264,-179.607,6.465,149.063
C06881=1144.901,67.582,-52.280,-179.604,6.466,149.063
C06882=1144.896,67.831,-52.296,-179.602,6.467,149.062
C06883=1144.892,68.080,-52.313,-179.599,6.469,149.062
C06884=1144.886,68.329,-52.330,-179.596,6.471,149.061
C06885=1144.881,68.579,-52.346,-179.594,6.471,149.061
C06886=1144.877,68.829,-52.362,-179.591,6.473,149.060
C06887=1144.871,69.077,-52.378,-179.588,6.474,149.060
C06888=1144.866,69.327,-52.396,-179.586,6.475,149.059
C06889=1144.861,69.576,-52.412,-179.583,6.477,149.059
C06890=1144.857,69.826,-52.429,-179.581,6.477,149.058
C06891=1144.852,70.075,-52.445,-179.578,6.479,149.058
C06892=1144.846,70.324,-52.462,-179.575,6.480,149.057
C06893=1144.842,70.574,-52.478,-179.573,6.481,149.057
C06894=1144.837,70.824,-52.495,-179.569,6.483,149.056
C06895=1144.831,71.073,-52.512,-179.567,6.484,149.056
C06896=1144.827,71.322,-52.528,-179.565,6.485,149.055
C06897=1144.822,71.572,-52.545,-179.562,6.487,149.055
C06898=1144.817,71.821,-52.562,-179.559,6.488,149.054
C06899=1144.812,72.070,-52.579,-179.556,6.489,149.054
C06900=1144.808,72.320,-52.595,-179.554,6.491,149.053
C06901=1144.802,72.569,-52.612,-179.550,6.492,149.053
C06902=1144.797,72.818,-52.629,-179.548,6.493,149.052
C06903=1144.793,73.068,-52.646,-179.546,6.494,149.052
C06904=1144.787,73.317,-52.662,-179.543,6.496,149.051
C06905=1144.783,73.566,-52.679,-179.540,6.496,149.051
C06906=1144.777,73.816,-52.696,-179.537,6.498,149.050
C06907=1144.772,74.065,-52.713,-179.535,6.500,149.050
C06908=1144.768,74.315,-52.729,-179.532,6.500,149.049
C06909=1144.763,74.564,-52.747,-179.529,6.502,149.049
C06910=1144.758,74.814,-52.763,-179.527,6.504,149.048
C06911=1144.752,75.063,-52.780,-179.524,6.504,149.048
C06912=1144.748,75.312,-52.797,-179.521,6.506,149.047
C06913=1144.743,75.562,-52.814,-179.518,6.507,149.047
C06914=1144.737,75.811,-52.830,-179.516,6.508,149.046
C06915=1144.733,76.060,-52.847,-179.513,6.510,149.046
C06916=1144.728,76.310,-52.865,-179.510,6.511,149.045
C06917=1144.724,76.559,-52.882,-179.508,6.513,149.045
C06918=1144.718,76.808,-52.899,-179.505,6.514,149.045
C06919=1144.713,77.058,-52.915,-179.502,6.515,149.044
C06920=1144.708,77.307,-52.933,-179.499,6.517,149.043
C06921=1144.704,77.557,-52.949,-179.497,6.518,149.043
C06922=1144.698,77.806,-52.966,-179.494,6.519,149.042
C06923=1144.694,78.055,-52.984,-179.491,6.521,149.042
C06924=1144.688,78.305,-53.001,-179.489,6.521,149.041
C06925=1144.684,78.554,-53.017,-179.486,6.523,149.041
C06926=1144.679,78.804,-53.035,-179.483,6.524,149.040
C06927=1144.674,79.053,-53.051,-179.481,6.526,149.040
C06928=1144.668,79.321,-53.070,-179.478,6.527,149.040
C06929=1144.663,79.590,-53.089,-179.475,6.528,149.039
C06930=1144.658,79.858,-53.107,-179.472,6.530,149.038
C06931=1144.652,80.127,-53.126,-179.469,6.531,149.038
C06932=1144.647,80.376,-53.143,-179.466,6.533,149.037
C06933=1144.643,80.625,-53.160,-179.464,6.534,149.037
C06934=1144.637,80.874,-53.177,-179.462,6.535,149.037
C06935=1144.633,81.124,-53.194,-179.458,6.537,149.036
C06936=1144.628,81.374,-53.211,-179.456,6.538,149.035
C06937=1144.623,81.623,-53.229,-179.453,6.540,149.035
C06938=1144.618,81.872,-53.246,-179.450,6.540,149.034
C06939=1144.613,82.122,-53.264,-179.447,6.542,149.034
C06940=1144.608,82.370,-53.280,-179.445,6.544,149.034
C06941=1144.603,82.620,-53.297,-179.442,6.545,149.033
C06942=1144.598,82.869,-53.315,-179.439,6.546,149.032
C06943=1144.594,83.119,-53.332,-179.437,6.548,149.032
C06944=1144.588,83.369,-53.349,-179.434,6.549,149.032
C06945=1144.583,83.618,-53.367,-179.432,6.550,149.031
C06946=1144.579,83.867,-53.384,-179.429,6.551,149.031
C06947=1144.574,84.116,-53.402,-179.426,6.553,149.030
C06948=1144.568,84.365,-53.419,-179.423,6.555,149.030
C06949=1144.564,84.614,-53.436,-179.421,6.556,149.029
C06950=1144.559,84.864,-53.453,-179.418,6.557,149.029
C06951=1144.554,85.113,-53.471,-179.415,6.559,149.028
C06952=1144.549,85.363,-53.489,-179.412,6.560,149.028
C06953=1144.545,85.612,-53.506,-179.410,6.561,149.027
C06954=1144.539,85.862,-53.523,-179.407,6.563,149.027
C06955=1144.534,86.111,-53.541,-179.404,6.564,149.026
C06956=1144.529,86.361,-53.558,-179.401,6.566,149.026
C06957=1144.525,86.610,-53.576,-179.399,6.568,149.025
C06958=1144.520,86.859,-53.593,-179.396,6.568,149.025
C06959=1144.515,87.109,-53.611,-179.393,6.570,149.024
C06960=1144.510,87.358,-53.628,-179.391,6.571,149.024
C06961=1144.505,87.607,-53.645,-179.388,6.573,149.024
C06962=1144.500,87.856,-53.663,-179.386,6.574,149.023
C06963=1144.495,88.106,-53.681,-179.382,6.575,149.022
C06964=1144.490,88.355,-53.699,-179.380,6.577,149.022
C06965=1144.485,88.604,-53.716,-179.377,6.579,149.022
C06966=1144.480,88.853,-53.733,-179.374,6.580,149.021
C06967=1144.476,89.103,-53.751,-179.372,6.581,149.021
C06968=1144.470,89.352,-53.769,-179.369,6.582,149.020
C06969=1144.465,89.601,-53.786,-179.366,6.584,149.020
C06970=1144.460,89.851,-53.804,-179.363,6.586,149.019
C06971=1144.455,90.100,-53.822,-179.361,6.587,149.019
C06972=1144.450,90.350,-53.840,-179.358,6.588,149.018
C06973=1144.446,90.598,-53.857,-179.355,6.590,149.018
C06974=1144.441,90.848,-53.874,-179.353,6.591,149.017
C06975=1144.436,91.097,-53.892,-179.350,6.593,149.017
C06976=1144.431,91.347,-53.910,-179.347,6.593,149.016
C06977=1144.426,91.596,-53.928,-179.344,6.595,149.016
C06978=1144.421,91.846,-53.946,-179.342,6.597,149.015
C06979=1144.417,92.095,-53.964,-179.339,6.598,149.015
C06980=1144.412,92.345,-53.982,-179.336,6.600,149.015
C06981=1144.407,92.594,-54.000,-179.334,6.601,149.014
C06982=1144.402,92.843,-54.018,-179.331,6.602,149.014
C06983=1144.397,93.093,-54.035,-179.328,6.604,149.013
C06984=1144.393,93.342,-54.053,-179.325,6.606,149.013
C06985=1144.388,93.591,-54.070,-179.323,6.607,149.012
C06986=1144.383,93.840,-54.088,-179.319,6.609,149.012
C06987=1144.378,94.089,-54.106,-179.317,6.610,149.011
C06988=1144.373,94.338,-54.124,-179.315,6.611,149.011
C06989=1144.368,94.588,-54.142,-179.312,6.613,149.010
C06990=1144.363,94.837,-54.160,-179.309,6.615,149.010
C06991=1144.358,95.087,-54.178,-179.306,6.616,149.009
C06992=1144.353,95.336,-54.196,-179.304,6.617,149.009
C06993=1144.349,95.586,-54.214,-179.301,6.618,149.008
C06994=1144.344,95.835,-54.232,-179.298,6.620,149.008
C06995=1144.339,96.084,-54.250,-179.296,6.622,149.008
C06996=1144.334,96.333,-54.268,-179.292,6.623,149.007
C06997=1144.329,96.582,-54.286,-179.290,6.625,149.007
C06998=1144.324,96.831,-54.304,-179.287,6.626,149.006
C06999=1144.318,97.081,-54.322,-179.285,6.627,149.006
C07000=1144.314,97.330,-54.340,-179.282,6.629,149.005
C07001=1144.309,97.580,-54.359,-179.279,6.630,149.005
C07002=1144.304,97.829,-54.377,-179.276,6.632,149.004
C07003=1144.299,98.078,-54.395,-179.273,6.634,149.004
C07004=1144.294,98.328,-54.413,-179.271,6.635,149.003
C07005=1144.290,98.577,-54.431,-179.268,6.636,149.003
C07006=1144.285,98.826,-54.449,-179.266,6.638,149.003
C07007=1144.280,99.076,-54.467,-179.262,6.639,149.002
C07008=1144.275,99.325,-54.485,-179.260,6.641,149.002
C07009=1144.270,99.574,-54.504,-179.257,6.643,149.001
C07010=1144.265,99.824,-54.522,-179.254,6.644,149.001
C07011=1144.260,100.073,-54.540,-179.252,6.646,149.000
C07012=1144.255,100.321,-54.558,-179.249,6.647,149.000
C07013=1144.251,100.571,-54.577,-179.246,6.648,148.999
C07014=1144.246,100.820,-54.595,-179.243,6.650,148.999
C07015=1144.241,101.070,-54.613,-179.241,6.651,148.998
C07016=1144.236,101.319,-54.631,-179.238,6.653,148.998
C07017=1144.231,101.569,-54.649,-179.235,6.655,148.998
C07018=1144.226,101.818,-54.667,-179.232,6.656,148.997
C07019=1144.222,102.067,-54.686,-179.229,6.658,148.997
C07020=1144.217,102.316,-54.704,-179.227,6.659,148.996
C07021=1144.211,102.565,-54.723,-179.224,6.660,148.996
C07022=1144.207,102.815,-54.741,-179.222,6.662,148.995
C07023=1144.202,103.064,-54.760,-179.219,6.664,148.995
C07024=1144.197,103.313,-54.778,-179.216,6.665,148.994
C07025=1144.192,103.562,-54.796,-179.213,6.667,148.994
C07026=1144.187,103.812,-54.815,-179.210,6.668,148.993
C07027=1144.183,104.061,-54.833,-179.208,6.670,148.993
C07028=1144.178,104.310,-54.851,-179.205,6.672,148.993
C07029=1144.173,104.560,-54.870,-179.202,6.674,148.992
C07030=1144.168,104.809,-54.889,-179.200,6.674,148.992
C07031=1144.163,105.058,-54.907,-179.197,6.676,148.991
C07032=1144.157,105.326,-54.927,-179.194,6.677,148.991
C07033=1144.153,105.595,-54.947,-179.191,6.680,148.990
C07034=1144.148,105.863,-54.967,-179.188,6.682,148.990
C07035=1144.142,106.132,-54.987,-179.185,6.683,148.989
C07036=1144.137,106.381,-55.005,-179.182,6.685,148.989
C07037=1144.133,106.630,-55.024,-179.179,6.686,148.988
C07038=1144.128,106.880,-55.042,-179.177,6.688,148.988
C07039=1144.122,107.129,-55.061,-179.174,6.690,148.988
C07040=1144.118,107.378,-55.080,-179.172,6.691,148.987
C07041=1144.113,107.627,-55.098,-179.169,6.692,148.987
C07042=1144.108,107.876,-55.117,-179.166,6.694,148.986
C07043=1144.104,108.126,-55.136,-179.163,6.695,148.986
C07044=1144.099,108.375,-55.154,-179.160,6.697,148.985
C07045=1144.093,108.624,-55.173,-179.158,6.699,148.985
C07046=1144.089,108.874,-55.192,-179.155,6.700,148.985
C07047=1144.084,109.123,-55.211,-179.152,6.702,148.984
C07048=1144.079,109.372,-55.229,-179.149,6.704,148.984
C07049=1144.075,109.621,-55.248,-179.146,6.705,148.983
C07050=1144.069,109.870,-55.267,-179.143,6.707,148.983
C07051=1144.065,110.120,-55.285,-179.141,6.708,148.982
C07052=1144.060,110.369,-55.305,-179.138,6.710,148.982
C07053=1144.055,110.618,-55.323,-179.135,6.712,148.981
C07054=1144.050,110.868,-55.342,-179.133,6.713,148.981
C07055=1144.046,111.116,-55.361,-179.130,6.714,148.981
C07056=1144.040,111.367,-55.380,-179.128,6.716,148.980
C07057=1144.036,111.615,-55.399,-179.124,6.717,148.980
C07058=1144.030,111.865,-55.417,-179.122,6.719,148.979
C07059=1144.026,112.114,-55.436,-179.119,6.721,148.979
C07060=1144.021,112.363,-55.455,-179.116,6.722,148.978
C07061=1144.017,112.613,-55.474,-179.114,6.724,148.978
C07062=1144.011,112.861,-55.493,-179.111,6.726,148.978
C07063=1144.007,113.111,-55.512,-179.108,6.727,148.977
C07064=1144.002,113.360,-55.531,-179.105,6.729,148.977
C07065=1143.997,113.609,-55.549,-179.103,6.731,148.976
C07066=1143.992,113.858,-55.569,-179.099,6.732,148.976
C07067=1143.987,114.108,-55.588,-179.097,6.734,148.975
C07068=1143.983,114.357,-55.607,-179.094,6.736,148.975
C07069=1143.977,114.606,-55.626,-179.091,6.737,148.974
C07070=1143.973,114.855,-55.645,-179.089,6.739,148.974
C07071=1143.968,115.105,-55.664,-179.086,6.741,148.974
C07072=1143.963,115.354,-55.683,-179.083,6.742,148.973
C07073=1143.958,115.603,-55.702,-179.080,6.744,148.973
C07074=1143.953,115.852,-55.722,-179.078,6.746,148.972
C07075=1143.949,116.101,-55.740,-179.075,6.747,148.972
C07076=1143.944,116.351,-55.759,-179.072,6.749,148.972
C07077=1143.938,116.600,-55.779,-179.069,6.750,148.971
C07078=1143.934,116.849,-55.798,-179.066,6.752,148.971
C07079=1143.929,117.098,-55.817,-179.064,6.754,148.970
C07080=1143.924,117.348,-55.837,-179.061,6.755,148.970
C07081=1143.920,117.596,-55.855,-179.058,6.757,148.969
C07082=1143.915,117.846,-55.875,-179.055,6.759,148.969
C07083=1143.909,118.095,-55.894,-179.053,6.761,148.969
C07084=1143.905,118.345,-55.913,-179.050,6.762,148.968
C07085=1143.900,118.593,-55.932,-179.047,6.764,148.968
C07086=1143.895,118.843,-55.952,-179.044,6.766,148.967
C07087=1143.891,119.093,-55.971,-179.042,6.767,148.967
C07088=1143.886,119.341,-55.990,-179.039,6.769,148.967
C07089=1143.881,119.591,-56.010,-179.036,6.771,148.966
C07090=1143.876,119.840,-56.029,-179.034,6.772,148.966
C07091=1143.872,120.089,-56.048,-179.030,6.774,148.965
C07092=1143.867,120.338,-56.067,-179.028,6.775,148.965
C07093=1143.862,120.587,-56.087,-179.025,6.777,148.964
C07094=1143.857,120.837,-56.106,-179.022,6.779,148.964
C07095=1143.852,121.085,-56.125,-179.019,6.780,148.964
C07096=1143.848,121.335,-56.145,-179.017,6.782,148.963
C07097=1143.842,121.584,-56.164,-179.014,6.784,148.963
C07098=1143.838,121.833,-56.184,-179.011,6.786,148.962
C07099=1143.833,122.083,-56.203,-179.009,6.787,148.962
C07100=1143.828,122.331,-56.222,-179.006,6.789,148.962
C07101=1143.823,122.581,-56.242,-179.003,6.791,148.961
C07102=1143.819,122.830,-56.262,-179.000,6.792,148.961
C07103=1143.814,123.079,-56.281,-178.998,6.794,148.960
C07104=1143.809,123.328,-56.301,-178.995,6.796,148.960
C07105=1143.804,123.578,-56.321,-178.992,6.797,148.960
C07106=1143.800,123.827,-56.339,-178.990,6.799,148.959
C07107=1143.795,124.076,-56.359,-178.987,6.801,148.959
C07108=1143.790,124.326,-56.379,-178.984,6.803,148.958
C07109=1143.785,124.574,-56.399,-178.981,6.805,148.958
C07110=1143.780,124.824,-56.418,-178.978,6.807,148.958
C07111=1143.776,125.073,-56.438,-178.975,6.808,148.957
C07112=1143.770,125.322,-56.457,-178.973,6.810,148.957
C07113=1143.766,125.572,-56.477,-178.969,6.811,148.956
C07114=1143.761,125.820,-56.497,-178.967,6.813,148.956
C07115=1143.756,126.069,-56.516,-178.964,6.815,148.955
C07116=1143.752,126.319,-56.536,-178.961,6.817,148.955
C07117=1143.747,126.568,-56.556,-178.959,6.818,148.955
C07118=1143.742,126.816,-56.575,-178.956,6.820,148.954
C07119=1143.737,127.066,-56.595,-178.953,6.822,148.954
C07120=1143.732,127.316,-56.615,-178.950,6.823,148.953
C07121=1143.728,127.565,-56.635,-178.948,6.825,148.953
C07122=1143.723,127.813,-56.654,-178.945,6.827,148.953
C07123=1143.718,128.063,-56.674,-178.942,6.828,148.952
C07124=1143.714,128.312,-56.694,-178.939,6.831,148.952
C07125=1143.709,128.561,-56.714,-178.936,6.833,148.951
C07126=1143.704,128.810,-56.734,-178.933,6.834,148.951
C07127=1143.699,129.059,-56.754,-178.931,6.836,148.951
C07128=1143.694,129.309,-56.773,-178.928,6.838,148.950
C07129=1143.690,129.558,-56.794,-178.925,6.839,148.950
C07130=1143.684,129.807,-56.813,-178.923,6.841,148.949
C07131=1143.680,130.056,-56.833,-178.920,6.843,148.949
C07132=1143.675,130.305,-56.853,-178.917,6.845,148.949
C07133=1143.671,130.555,-56.873,-178.914,6.846,148.948
C07134=1143.665,130.804,-56.894,-178.912,6.848,148.948
C07135=1143.660,131.053,-56.913,-178.908,6.850,148.947
C07136=1143.655,131.321,-56.935,-178.906,6.852,148.947
C07137=1143.650,131.590,-56.956,-178.903,6.854,148.947
C07138=1143.645,131.859,-56.978,-178.900,6.856,148.946
C07139=1143.640,132.127,-56.999,-178.897,6.858,148.946
C07140=1143.635,132.376,-57.020,-178.894,6.860,148.945
C07141=1143.630,132.625,-57.040,-178.891,6.862,148.945
C07142=1143.626,132.875,-57.060,-178.889,6.863,148.945
C07143=1143.621,133.124,-57.080,-178.886,6.865,148.944
C07144=1143.616,133.373,-57.099,-178.883,6.867,148.944
C07145=1143.611,133.622,-57.120,-178.880,6.869,148.943
C07146=1143.607,133.871,-57.140,-178.877,6.871,148.943
C07147=1143.601,134.121,-57.160,-178.875,6.873,148.943
C07148=1143.597,134.369,-57.181,-178.872,6.874,148.942
C07149=1143.593,134.618,-57.201,-178.869,6.876,148.942
C07150=1143.588,134.868,-57.221,-178.866,6.878,148.941
C07151=1143.583,135.116,-57.241,-178.864,6.879,148.941
C07152=1143.578,135.365,-57.262,-178.860,6.882,148.941
C07153=1143.573,135.615,-57.281,-178.858,6.884,148.940
C07154=1143.568,135.864,-57.302,-178.855,6.885,148.940
C07155=1143.564,136.113,-57.322,-178.852,6.887,148.940
C07156=1143.559,136.363,-57.342,-178.850,6.889,148.939
C07157=1143.554,136.612,-57.363,-178.847,6.890,148.939
C07158=1143.550,136.861,-57.383,-178.844,6.892,148.938
C07159=1143.545,137.110,-57.403,-178.841,6.895,148.938
C07160=1143.540,137.360,-57.424,-178.838,6.896,148.938
C07161=1143.535,137.608,-57.444,-178.835,6.898,148.937
C07162=1143.530,137.857,-57.464,-178.833,6.900,148.937
C07163=1143.526,138.106,-57.484,-178.830,6.901,148.936
C07164=1143.521,138.355,-57.505,-178.828,6.903,148.936
C07165=1143.516,138.605,-57.525,-178.824,6.906,148.936
C07166=1143.511,138.853,-57.545,-178.822,6.908,148.935
C07167=1143.506,139.103,-57.566,-178.819,6.909,148.935
C07168=1143.502,139.352,-57.587,-178.816,6.911,148.935
C07169=1143.497,139.601,-57.607,-178.814,6.913,148.934
C07170=1143.492,139.850,-57.628,-178.811,6.915,148.934
C07171=1143.488,140.099,-57.649,-178.807,6.917,148.934
C07172=1143.483,140.348,-57.668,-178.805,6.919,148.933
C07173=1143.478,140.598,-57.689,-178.802,6.920,148.933
C07174=1143.473,140.847,-57.709,-178.799,6.922,148.932
C07175=1143.468,141.096,-57.730,-178.797,6.924,148.932
C07176=1143.464,141.345,-57.751,-178.794,6.926,148.932
C07177=1143.459,141.594,-57.771,-178.791,6.928,148.931
C07178=1143.454,141.843,-57.792,-178.788,6.930,148.931
C07179=1143.450,142.092,-57.813,-178.786,6.932,148.931
C07180=1143.445,142.341,-57.834,-178.783,6.934,148.930
C07181=1143.440,142.590,-57.854,-178.780,6.935,148.930
C07182=1143.435,142.839,-57.875,-178.777,6.938,148.930
C07183=1143.431,143.088,-57.895,-178.774,6.940,148.929
C07184=1143.426,143.337,-57.916,-178.771,6.941,148.929
C07185=1143.421,143.587,-57.937,-178.769,6.943,148.928
C07186=1143.417,143.836,-57.957,-178.766,6.945,148.928
C07187=1143.411,144.085,-57.978,-178.763,6.947,148.928
C07188=1143.408,144.334,-57.999,-178.760,6.949,148.927
C07189=1143.403,144.583,-58.020,-178.757,6.951,148.927
C07190=1143.398,144.832,-58.041,-178.755,6.953,148.927
C07191=1143.393,145.081,-58.062,-178.752,6.954,148.926
C07192=1143.389,145.330,-58.082,-178.749,6.957,148.926
C07193=1143.383,145.580,-58.103,-178.746,6.959,148.926
C07194=1143.379,145.828,-58.123,-178.744,6.960,148.925
C07195=1143.374,146.078,-58.144,-178.741,6.962,148.925
C07196=1143.369,146.326,-58.166,-178.738,6.964,148.924
C07197=1143.364,146.575,-58.186,-178.735,6.966,148.924
C07198=1143.359,146.825,-58.207,-178.732,6.968,148.924
C07199=1143.355,147.074,-58.228,-178.730,6.970,148.923
C07200=1143.350,147.324,-58.249,-178.727,6.972,148.923
C07201=1143.345,147.572,-58.271,-178.724,6.974,148.923
C07202=1143.341,147.821,-58.291,-178.721,6.976,148.922
C07203=1143.336,148.070,-58.312,-178.719,6.978,148.922
C07204=1143.332,148.319,-58.333,-178.716,6.979,148.922
C07205=1143.327,148.568,-58.354,-178.713,6.982,148.921
C07206=1143.322,148.818,-58.375,-178.710,6.984,148.921
C07207=1143.318,149.067,-58.396,-178.708,6.986,148.921
C07208=1143.313,149.315,-58.418,-178.705,6.987,148.920
C07209=1143.307,149.565,-58.438,-178.702,6.990,148.920
C07210=1143.303,149.814,-58.459,-178.699,6.992,148.919
C07211=1143.298,150.062,-58.481,-178.696,6.993,148.919
C07212=1143.294,150.312,-58.502,-178.693,6.995,148.919
C07213=1143.289,150.561,-58.523,-178.690,6.998,148.918
C07214=1143.284,150.810,-58.544,-178.688,7.000,148.918
C07215=1143.279,151.059,-58.565,-178.685,7.001,148.918
C07216=1143.275,151.307,-58.586,-178.682,7.003,148.917
C07217=1143.270,151.557,-58.607,-178.679,7.006,148.917
C07218=1143.266,151.806,-58.629,-178.676,7.007,148.917
C07219=1143.260,152.055,-58.650,-178.674,7.009,148.916
C07220=1143.256,152.304,-58.671,-178.671,7.011,148.916
C07221=1143.251,152.553,-58.692,-178.668,7.014,148.916
C07222=1143.246,152.803,-58.713,-178.666,7.015,148.915
C07223=1143.242,153.052,-58.735,-178.663,7.017,148.915
C07224=1143.236,153.301,-58.756,-178.660,7.019,148.915
C07225=1143.232,153.549,-58.777,-178.657,7.021,148.914
C07226=1143.228,153.798,-58.799,-178.654,7.023,148.914
C07227=1143.223,154.048,-58.820,-178.652,7.025,148.914
C07228=1143.218,154.296,-58.842,-178.649,7.028,148.913
C07229=1143.213,154.546,-58.863,-178.646,7.029,148.913
C07230=1143.209,154.795,-58.884,-178.643,7.031,148.913
C07231=1143.204,155.044,-58.905,-178.640,7.033,148.912
C07232=1143.199,155.293,-58.927,-178.637,7.035,148.912
C07233=1143.195,155.542,-58.949,-178.635,7.037,148.912
C07234=1143.190,155.791,-58.970,-178.632,7.039,148.911
C07235=1143.185,156.040,-58.992,-178.629,7.042,148.911
C07236=1143.180,156.288,-59.013,-178.626,7.043,148.911
C07237=1143.176,156.538,-59.034,-178.623,7.045,148.910
C07238=1143.171,156.787,-59.056,-178.621,7.048,148.910
C07239=1143.166,157.035,-59.077,-178.618,7.050,148.910
C07240=1143.161,157.305,-59.101,-178.615,7.051,148.909
C07241=1143.156,157.574,-59.123,-178.612,7.054,148.909
C07242=1143.151,157.843,-59.147,-178.609,7.056,148.909
C07243=1143.146,158.112,-59.170,-178.606,7.058,148.908
C07244=1143.142,158.361,-59.192,-178.603,7.060,148.908
C07245=1143.137,158.610,-59.213,-178.600,7.062,148.907
C07246=1143.132,158.859,-59.235,-178.598,7.064,148.907
C07247=1143.128,159.108,-59.257,-178.595,7.066,148.907
C07248=1143.123,159.357,-59.279,-178.592,7.069,148.907
C07249=1143.118,159.605,-59.300,-178.589,7.070,148.906
C07250=1143.113,159.855,-59.322,-178.586,7.072,148.906
C07251=1143.109,160.104,-59.343,-178.583,7.075,148.906
C07252=1143.104,160.353,-59.365,-178.581,7.077,148.905
C07253=1143.099,160.602,-59.387,-178.578,7.078,148.905
C07254=1143.095,160.851,-59.409,-178.575,7.081,148.905
C07255=1143.090,161.100,-59.431,-178.573,7.083,148.904
C07256=1143.085,161.349,-59.453,-178.570,7.085,148.904
C07257=1143.081,161.599,-59.474,-178.567,7.087,148.904
C07258=1143.076,161.847,-59.496,-178.564,7.089,148.903
C07259=1143.071,162.096,-59.517,-178.562,7.091,148.903
C07260=1143.067,162.345,-59.539,-178.558,7.094,148.903
C07261=1143.062,162.594,-59.561,-178.556,7.095,148.902
C07262=1143.058,162.843,-59.583,-178.553,7.097,148.902
C07263=1143.052,163.092,-59.605,-178.550,7.100,148.902
C07264=1143.048,163.341,-59.627,-178.547,7.102,148.901
C07265=1143.043,163.590,-59.649,-178.544,7.104,148.901
C07266=1143.039,163.839,-59.671,-178.541,7.106,148.901
C07267=1143.034,164.088,-59.693,-178.539,7.108,148.900
C07268=1143.030,164.337,-59.715,-178.536,7.111,148.900
C07269=1143.025,164.586,-59.737,-178.533,7.112,148.900
C07270=1143.020,164.835,-59.759,-178.530,7.114,148.899
C07271=1143.015,165.084,-59.781,-178.527,7.117,148.899
C07272=1143.011,165.334,-59.803,-178.525,7.119,148.899
C07273=1143.006,165.582,-59.825,-178.522,7.120,148.899
C07274=1143.002,165.831,-59.847,-178.519,7.123,148.898
C07275=1142.997,166.080,-59.869,-178.517,7.125,148.898
C07276=1142.993,166.329,-59.891,-178.513,7.128,148.898
C07277=1142.987,166.578,-59.913,-178.511,7.129,148.897
C07278=1142.983,166.827,-59.935,-178.508,7.131,148.897
C07279=1142.978,167.076,-59.957,-178.505,7.134,148.897
C07280=1142.974,167.325,-59.980,-178.502,7.136,148.896
C07281=1142.968,167.574,-60.002,-178.499,7.138,148.896
C07282=1142.964,167.823,-60.024,-178.496,7.140,148.896
C07283=1142.959,168.072,-60.046,-178.494,7.142,148.896
C07284=1142.955,168.321,-60.068,-178.491,7.144,148.895
C07285=1142.950,168.569,-60.091,-178.488,7.146,148.895
C07286=1142.945,168.819,-60.113,-178.486,7.148,148.895
C07287=1142.941,169.068,-60.135,-178.483,7.151,148.894
C07288=1142.935,169.317,-60.157,-178.480,7.153,148.894
C07289=1142.931,169.566,-60.180,-178.477,7.155,148.894
C07290=1142.927,169.814,-60.202,-178.475,7.157,148.893
C07291=1142.922,170.064,-60.224,-178.471,7.160,148.893
C07292=1142.917,170.312,-60.247,-178.469,7.161,148.893
C07293=1142.913,170.561,-60.269,-178.466,7.163,148.893
C07294=1142.908,170.811,-60.291,-178.463,7.166,148.892
C07295=1142.903,171.059,-60.314,-178.460,7.168,148.892
C07296=1142.899,171.308,-60.336,-178.457,7.171,148.892
C07297=1142.894,171.557,-60.359,-178.455,7.172,148.891
C07298=1142.889,171.806,-60.381,-178.452,7.174,148.891
C07299=1142.885,172.055,-60.403,-178.449,7.177,148.891
C07300=1142.880,172.304,-60.426,-178.447,7.179,148.891
C07301=1142.875,172.553,-60.448,-178.443,7.181,148.890
C07302=1142.871,172.802,-60.471,-178.441,7.183,148.890
C07303=1142.866,173.051,-60.493,-178.438,7.186,148.890
C07304=1142.862,173.299,-60.516,-178.435,7.188,148.889
C07305=1142.857,173.549,-60.538,-178.432,7.189,148.889
C07306=1142.852,173.797,-60.561,-178.430,7.192,148.889
C07307=1142.847,174.047,-60.584,-178.427,7.194,148.888
C07308=1142.843,174.295,-60.606,-178.424,7.196,148.888
C07309=1142.838,174.544,-60.629,-178.421,7.199,148.888
C07310=1142.834,174.793,-60.651,-178.418,7.201,148.888
C07311=1142.829,175.043,-60.674,-178.416,7.203,148.887
C07312=1142.824,175.291,-60.696,-178.413,7.206,148.887
C07313=1142.819,175.540,-60.719,-178.410,7.207,148.887
C07314=1142.815,175.789,-60.742,-178.408,7.210,148.887
C07315=1142.811,176.038,-60.765,-178.404,7.212,148.886
C07316=1142.806,176.287,-60.787,-178.402,7.214,148.886
C07317=1142.801,176.536,-60.810,-178.399,7.217,148.886
C07318=1142.797,176.785,-60.833,-178.396,7.218,148.885
C07319=1142.792,177.034,-60.856,-178.393,7.221,148.885
C07320=1142.788,177.282,-60.878,-178.391,7.223,148.885
C07321=1142.783,177.531,-60.901,-178.387,7.226,148.885
C07322=1142.778,177.781,-60.924,-178.385,7.227,148.884
C07323=1142.774,178.030,-60.947,-178.382,7.230,148.884
C07324=1142.769,178.278,-60.970,-178.379,7.232,148.884
C07325=1142.764,178.527,-60.992,-178.376,7.235,148.884
C07326=1142.760,178.776,-61.015,-178.374,7.237,148.883
C07327=1142.756,179.025,-61.038,-178.370,7.239,148.883
C07328=1142.750,179.273,-61.061,-178.368,7.241,148.883
C07329=1142.745,179.523,-61.084,-178.365,7.243,148.882
C07330=1142.741,179.772,-61.106,-178.362,7.245,148.882
C07331=1142.737,180.021,-61.130,-178.360,7.248,148.882
